// TwinCAT 3 PLC project Gearsim
// ProgramVersion: 3.1.4023.0
// libraries:
//   Struckig, * (Stefan Besler)
//   Tc3_Module, * (Beckhoff Automation GmbH)
//   ZApplication, 1.5.38.0 (Zeugwerk GmbH)
//   ZEquipment, 1.5.38.0 (Zeugwerk GmbH)
//   ZAux, 1.5.38.0 (Zeugwerk GmbH)
//   ZPlatform, 1.5.38.0 (Zeugwerk GmbH)
//   ZCore, 1.5.38.0 (Zeugwerk GmbH)
// project tree:
//   ZApp/App/ ZApp.TcPOU
//   ZApp/App/_DataTypes/ ZAppStep.TcDUT
//   ZApp/App/_States/ ZAppSequenceBoot.TcPOU, ZAppSequenceBootFault.TcPOU, ZAppSequenceRunning.TcPOU
//   ZApp/App/_SubObjects/ ZAppSequence.TcPOU
//   ZApp/Com/_DataTypes/ ZCom.TcDUT, ZComUnit.TcDUT
//   ZApp/Data/_DataTypes/ ZData.TcDUT, ZDataMachine.TcDUT, ZDataConfig.TcDUT, ZDataCalibration.TcDUT, ZDataRecipe.TcDUT
//   ZApp/Unit/Gear/ GearUnit.TcPOU, GearUnitProgram.TcPOU, IGear.TcIO
//   ZApp/Unit/Gear/_Com/ GearCom.TcDUT, GearComPublish.TcDUT, GearComPublishEquipment.TcDUT, GearComRef.TcDUT, GearComRequest.TcDUT, GearComSubscribe.TcDUT, GearComSubscribeEquipment.TcDUT
//   ZApp/Unit/Gear/_DataTypes/ GearRole.TcDUT, GearState.TcDUT, GearStep.TcDUT
//   ZApp/Unit/Gear/_Data/ GearDataCalibration.TcDUT, GearDataConfig.TcDUT, GearDataMachine.TcDUT, GearDataRef.TcDUT
//   ZApp/Unit/Gear/_Equipment/ GearActuator.TcPOU, GearAxis.TcPOU, GearEquipment.TcPOU, GearFieldbus.TcPOU, GearIo.TcPOU, GearLinkedUnit.TcPOU
//   ZApp/Unit/Gear/_States/ GearSequenceAutomatic.TcPOU, GearSequenceBoot.TcPOU, GearSequenceFaultReaction.TcPOU, GearSequenceGoHome.TcPOU, GearSequenceStop.TcPOU
//   ZApp/Unit/Gear/_SubObjects/ GearContainer.TcPOU, GearSequence.TcPOU
//   ZApp/Unit/Gear/_SubSequences/ GearSequenceAutomaticPrimary.TcPOU, GearSequenceAutomaticSecondarySimple.TcPOU, GearSequenceAutomaticSecondaryStruckig.TcPOU, GearSubSequence.TcPOU
//   ZApp/Unit/Machine/ IMachine.TcIO, MachineUnit.TcPOU, MachineUnitProgram.TcPOU
//   ZApp/Unit/Machine/_Com/ MachineCom.TcDUT, MachineComPublish.TcDUT, MachineComPublishEquipment.TcDUT, MachineComRef.TcDUT, MachineComRequest.TcDUT, MachineComSubscribe.TcDUT, MachineComSubscribeEquipment.TcDUT
//   ZApp/Unit/Machine/_DataTypes/ MachineState.TcDUT, MachineStep.TcDUT
//   ZApp/Unit/Machine/_Data/ MachineDataCalibration.TcDUT, MachineDataConfig.TcDUT, MachineDataMachine.TcDUT, MachineDataRef.TcDUT
//   ZApp/Unit/Machine/_Equipment/ MachineActuator.TcPOU, MachineAxis.TcPOU, MachineEquipment.TcPOU, MachineFieldbus.TcPOU, MachineIo.TcPOU, MachineLinkedUnit.TcPOU
//   ZApp/Unit/Machine/_States/ MachineSequenceAutomatic.TcPOU, MachineSequenceBoot.TcPOU, MachineSequenceFaultReaction.TcPOU, MachineSequenceGoHome.TcPOU, MachineSequenceStop.TcPOU
//   ZApp/Unit/Machine/_SubObjects/ MachineContainer.TcPOU, MachineSequence.TcPOU
//   ZApp/ ZGlobal.TcGVL, ZModuleProgram.TcPOU, ZModuleTask.TcTTO
// real-time tasks:
//   TASK ZModuleTask: cycle T#10ms, priority 20, ADS port 350
//   TASK ZModuleTask1: cycle T#10ms, priority 21, ADS port 351

CONFIGURATION Gearsim
    RESOURCE PLC ON TwinCAT3
        TASK ZModuleTask(INTERVAL := T#10ms, PRIORITY := 21);
        PROGRAM ZModuleProgram WITH ZModuleTask : ZModuleProgram;
    END_RESOURCE
END_CONFIGURATION

// ---- ZApp/App/_DataTypes/ZAppStep.TcDUT
{attribute 'qualified_only'}
{attribute 'to_string'}
TYPE ZAppStep :
(
  Undefined := 0
  
  ,BootBegin
  ,BootLoadDefaultData
  ,BootEnd
  ,BootFaultBegin
  ,BootFaultEnd 
  ,RunningBegin
  ,RunningEnd   
);
END_TYPE

// ---- ZApp/Com/_DataTypes/ZCom.TcDUT
TYPE ZCom :
STRUCT
  // module context
  App : ZApplication.ApplicationComPublish;
  Alarming : ZApplication.AlarmingCom;
  Messages : ZApplication.MessagingCom;
  
  // unit context
  Unit : ZComUnit;

END_STRUCT
END_TYPE

// ---- ZApp/Com/_DataTypes/ZComUnit.TcDUT
TYPE ZComUnit :
STRUCT
{region "LeftGear"}
{IF NOT (defined (LeftGear_disabled))}
  LeftGear : GearCom;
  {attribute 'ZId' := 'd1deea68-6f8b-4ea5-9916-7be69dc951fa'}
{END_IF}
{endregion}
{region "Machine"}
{IF NOT (defined (Machine_disabled))}
  Machine : MachineCom;
  {attribute 'ZId' := '9a1e8940-043c-4b8f-bd95-526fb267b71c'}
{END_IF}
{endregion}
{region "RightGear"}
{IF NOT (defined (RightGear_disabled))}
  RightGear : GearCom;
  {attribute 'ZId' := '215d1db4-d61a-4f46-91b5-612373b86c91'}
{END_IF}
{endregion}
{attribute '__ZwPlcApplicationComUnitDeclaration__'} // Do not remove this attribute! It is used for code generation.
END_STRUCT
END_TYPE

// ---- ZApp/Data/_DataTypes/ZData.TcDUT
TYPE ZData :
STRUCT
  Config : ZDataConfig;
  Machine : ZDataMachine;
  Calibration : ZDataCalibration;
  Recipe : ZDataRecipe;
END_STRUCT
END_TYPE

// ---- ZApp/Data/_DataTypes/ZDataMachine.TcDUT
TYPE ZDataMachine :
STRUCT
{region "PrimaryGear"}
{IF NOT (defined (PrimaryGear_disabled))}
  PrimaryGear : GearDataMachine;
  {attribute 'ZId' := 'd1deea68-6f8b-4ea5-9916-7be69dc951fa'}
{END_IF}
{endregion}
{region "Machine"}
{IF NOT (defined (Machine_disabled))}
  Machine : MachineDataMachine;
  {attribute 'ZId' := '9a1e8940-043c-4b8f-bd95-526fb267b71c'}
{END_IF}
{endregion}
{region "SimpleGear"}
{IF NOT (defined (SimpleGear_disabled))}
  SimpleGear : GearDataMachine;
  {attribute 'ZId' := '215d1db4-d61a-4f46-91b5-612373b86c91'}
{END_IF}
{endregion}
{region "StruckigGear"}
{IF NOT (defined (StruckigGear_disabled))}
  StruckigGear : GearDataMachine;
  {attribute 'ZId' := 'd827270e-999f-436d-80d5-b12442f5d1cf'}
{END_IF}
{endregion}
{attribute '__ZwPlcApplicationDataMachineDeclaration__'} // Do not remove this attribute! It is used for code generation.
END_STRUCT
END_TYPE

// ---- ZApp/Data/_DataTypes/ZDataConfig.TcDUT
TYPE ZDataConfig :
STRUCT
{region "PrimaryGear"}
{IF NOT (defined (PrimaryGear_disabled))}
  PrimaryGear : GearDataConfig;
  {attribute 'ZId' := 'd1deea68-6f8b-4ea5-9916-7be69dc951fa'}
{END_IF}
{endregion}
{region "Machine"}
{IF NOT (defined (Machine_disabled))}
  Machine : MachineDataConfig;
  {attribute 'ZId' := '9a1e8940-043c-4b8f-bd95-526fb267b71c'}
{END_IF}
{endregion}
{region "SimpleGear"}
{IF NOT (defined (SimpleGear_disabled))}
  SimpleGear : GearDataConfig;
  {attribute 'ZId' := '215d1db4-d61a-4f46-91b5-612373b86c91'}
{END_IF}
{endregion}
{region "StruckigGear"}
{IF NOT (defined (StruckigGear_disabled))}
  StruckigGear : GearDataConfig;
  {attribute 'ZId' := 'd827270e-999f-436d-80d5-b12442f5d1cf'}
{END_IF}
{endregion}
{attribute '__ZwPlcApplicationDataConfigDeclaration__'} // Do not remove this attribute! It is used for code generation.
END_STRUCT
END_TYPE

// ---- ZApp/Data/_DataTypes/ZDataCalibration.TcDUT
TYPE ZDataCalibration :
STRUCT
{region "PrimaryGear"}
{IF NOT (defined (PrimaryGear_disabled))}
  PrimaryGear : GearDataCalibration;
  {attribute 'ZId' := 'd1deea68-6f8b-4ea5-9916-7be69dc951fa'}
{END_IF}
{endregion}
{region "Machine"}
{IF NOT (defined (Machine_disabled))}
  Machine : MachineDataCalibration;
  {attribute 'ZId' := '9a1e8940-043c-4b8f-bd95-526fb267b71c'}
{END_IF}
{endregion}
{region "SimpleGear"}
{IF NOT (defined (SimpleGear_disabled))}
  SimpleGear : GearDataCalibration;
  {attribute 'ZId' := '215d1db4-d61a-4f46-91b5-612373b86c91'}
{END_IF}
{endregion}
{region "StruckigGear"}
{IF NOT (defined (StruckigGear_disabled))}
  StruckigGear : GearDataCalibration;
  {attribute 'ZId' := 'd827270e-999f-436d-80d5-b12442f5d1cf'}
{END_IF}
{endregion}
{attribute '__ZwPlcApplicationDataCalibrationDeclaration__'} // Do not remove this attribute! It is used for code generation.
END_STRUCT
END_TYPE

// ---- ZApp/Data/_DataTypes/ZDataRecipe.TcDUT
TYPE ZDataRecipe :
STRUCT
  RecipeParam1 : LREAL;
  RecipeParam2 : LREAL;
  RecipeParam3 : LREAL;
END_STRUCT
END_TYPE

// ---- ZApp/Unit/Gear/_Com/GearCom.TcDUT
/// This struct contains variables that
/// * are read from outside (e.g. HMI) to retrieve information about the unit's current state and (temporary) parameters (= `publish`) 
/// * are written from outside (e.g. HMI) to control the unit via ADS (= `subscribe`) 
TYPE GearCom :
STRUCT
  Publish : GearComPublish;
  Subscribe : GearComSubscribe;
END_STRUCT
END_TYPE

// ---- ZApp/Unit/Gear/_Com/GearComPublish.TcDUT
/// this is the container of informations that the unit wants to share with the world outside of the PLC
/// This struct should only be read from by external applications.
TYPE GearComPublish :
STRUCT
  State : ZApplication.UnitStateMachineState; // state the unit is in
  Request : GearComRequest; // booleans that indictate which action is currently possible to perform with this unit
  Equipment : GearComPublishEquipment;  // structs for equipment objects which are used by the bridges
END_STRUCT
END_TYPE

// ---- ZApp/Unit/Gear/_Com/GearComPublishEquipment.TcDUT
TYPE GearComPublishEquipment :
STRUCT

{region "PositionX : Axis"}
  PositionX : ZApplication.AxisComPublish;
  {attribute 'ZId' := 'fbe544fd-32f7-4a35-b34a-168d60744a34'}
{endregion}

{region "RotationC : Axis"}
  RotationC : ZApplication.AxisComPublish;
  {attribute 'ZId' := '01f1af52-e172-4e11-895e-2a66564d7b35'}
{endregion}

{attribute '__ZwPlcUnitComDeclaration__'} // Do not remove this attribute! It is used for code generation.

END_STRUCT
END_TYPE

// ---- ZApp/Unit/Gear/_Com/GearComRef.TcDUT
/// container for all communication data types that are used by the unit
TYPE GearComRef :
STRUCT
  Publish : REFERENCE TO GearComPublish; 
  Subscribe : REFERENCE TO GearComSubscribe; 
END_STRUCT
END_TYPE

// ---- ZApp/Unit/Gear/_Com/GearComRequest.TcDUT
TYPE GearComRequest :
STRUCT
  Start : BOOL;
  Stop : BOOL;
  GoHome : BOOL;
  Halt : BOOL;
END_STRUCT
END_TYPE

// ---- ZApp/Unit/Gear/_Com/GearComSubscribe.TcDUT
TYPE GearComSubscribe :
STRUCT
  Request : GearComRequest; // contains booleans that are used to start a specific sequence.
  Equipment : GearComSubscribeEquipment;  // structs for equipment objects which are used by the bridges
END_STRUCT
END_TYPE

// ---- ZApp/Unit/Gear/_Com/GearComSubscribeEquipment.TcDUT
TYPE GearComSubscribeEquipment :
STRUCT

{region "PositionX : Axis"}
  PositionX : ZApplication.AxisComSubscribe;
  {attribute 'ZId' := 'fbe544fd-32f7-4a35-b34a-168d60744a34'}
{endregion}

{region "RotationC : Axis"}
  RotationC : ZApplication.AxisComSubscribe;
  {attribute 'ZId' := '01f1af52-e172-4e11-895e-2a66564d7b35'}
{endregion}

{attribute '__ZwPlcUnitComDeclaration__'} // Do not remove this attribute! It is used for code generation.

END_STRUCT
END_TYPE

// ---- ZApp/Unit/Gear/_DataTypes/GearRole.TcDUT
{attribute 'qualified_only'}
{attribute 'strict'}
TYPE GearRole :
(
  Undefined
	,Primary
  ,SecondarySimple
  ,SecondaryStruckig
);
END_TYPE

// ---- ZApp/Unit/Gear/_DataTypes/GearState.TcDUT
/// This enumeration contains all used defined sequences of a unit.
/// Per default a unit makes use of the states that are contained in (UnitStateDefault)[xref:ZApplication.UnitStateDefault]. However,
/// most of the time a unit need to perform some application depend sequences that can be performed by putting the unit into userdefined states.
/// For instance, a robotic unit could use the state (automatic)[xref:ZApplication.UnitStateDefault] to lift an object from point A to point B,
/// a userdefined state could be used to open and close the robotic-units gripper, respectively
{attribute 'qualified_only'}
TYPE GearState :
(
	UserdefinedState1 := ZApplication.UnitStateMachineState.Last+1
);
END_TYPE

// ---- ZApp/Unit/Gear/_DataTypes/GearStep.TcDUT
/// This enumeration contains all steps that are used by the various sequences of a unit.
/// Sequences use a subrange (***Begin to ***End) of this enumeration.
{attribute 'qualified_only'}
{attribute 'to_string'}
TYPE GearStep :
(
  Undefined := 0
  
  ,BootBegin
  ,BootEnd 

  ,StopBegin
  ,StopEnd

  ,AutomaticBegin
  ,AutomaticEnd
  
  ,GoHomeBegin
  ,GoHomePositionX
  ,GoHomeRotationC
  ,GoHomeEnd 
  
  ,FaultReactionBegin
  ,FaultReactionEnd
  ,AutomaticPrimaryBegin
  ,AutomaticPrimaryHalt  
  ,AutomaticPrimaryEnd
  
  ,AutomaticSecondarySimpleBegin
  ,AutomaticSecondarySimpleCloseGap
  ,AutomaticSecondarySimpleSynchronized
  ,AutomaticSecondarySimpleOpenGap
  ,AutomaticSecondarySimpleTearDown
  ,AutomaticSecondarySimpleSpinFast
  ,AutomaticSecondarySimpleSpin
  ,AutomaticSecondarySimpleHalt    
  ,AutomaticSecondarySimpleEnd
  
  ,AutomaticSecondaryStruckigBegin
  ,AutomaticSecondaryStruckigRotate
  ,AutomaticSecondaryStruckigCloseGap
  ,AutomaticSecondaryStruckigSynchronized
  ,AutomaticSecondaryStruckigOpenGap
  ,AutomaticSecondaryStruckigTearDown
  ,AutomaticSecondaryStruckigSpinFast
  ,AutomaticSecondaryStruckigSpin
  ,AutomaticSecondaryStruckigHalt     
  ,AutomaticSecondaryStruckigEnd
);
END_TYPE

// ---- ZApp/Unit/Gear/_Data/GearDataCalibration.TcDUT
/// calibration that is determined by calibration sequences of the unit (static offsets, shifts)
TYPE GearDataCalibration :
STRUCT
  OffsetRotationC : LREAL;
END_STRUCT
END_TYPE

// ---- ZApp/Unit/Gear/_Data/GearDataConfig.TcDUT
/// configuration data that is used during boot to configure the Units equipment
TYPE GearDataConfig :
STRUCT
  Simulated : BOOL;
END_STRUCT
END_TYPE

// ---- ZApp/Unit/Gear/_Data/GearDataMachine.TcDUT
/// machine data that is used through most sequences of the unit (motor speed, axes positions, ...)
TYPE GearDataMachine :
STRUCT
  Role : GearRole;
  SlowspeedX : LREAL;
  HighspeedX : LREAL;
  HomePositionX : LREAL;
  SafePositionX : LREAL;
  SpinPositionX : LREAL;
  
  SlowspeedC : LREAL;
  HighspeedC : LREAL;  
  HomeRotationC : LREAL;
  
  ToothAngle : LREAL;
END_STRUCT
END_TYPE

// ---- ZApp/Unit/Gear/_Data/GearDataRef.TcDUT
/// container for all data that are used by the unit
TYPE GearDataRef :
STRUCT
  Config : REFERENCE TO GearDataConfig; // data required for booting the unit (axes configuration, simulation, parameters that have to be written in PREOP, ...)
  Machine : REFERENCE TO GearDataMachine; // speeds, positions, ...
  Calibration : REFERENCE TO GearDataCalibration; // offsets, shifts of nominal to actual values
END_STRUCT
END_TYPE

// ---- ZApp/Unit/Machine/_Com/MachineCom.TcDUT
/// This struct contains variables that
/// * are read from outside (e.g. HMI) to retrieve information about the unit's current state and (temporary) parameters (= `publish`) 
/// * are written from outside (e.g. HMI) to control the unit via ADS (= `subscribe`) 
TYPE MachineCom :
STRUCT
  Publish : MachineComPublish;
  Subscribe : MachineComSubscribe;
END_STRUCT
END_TYPE

// ---- ZApp/Unit/Machine/_Com/MachineComPublish.TcDUT
/// this is the container of informations that the unit wants to share with the world outside of the PLC
/// This struct should only be read from by external applications.
TYPE MachineComPublish :
STRUCT
  State : ZApplication.UnitStateMachineState; // state the unit is in
  Request : MachineComRequest; // booleans that indictate which action is currently possible to perform with this unit
  Equipment : MachineComPublishEquipment;  // structs for equipment objects which are used by the bridges
END_STRUCT
END_TYPE

// ---- ZApp/Unit/Machine/_Com/MachineComPublishEquipment.TcDUT
TYPE MachineComPublishEquipment :
STRUCT

{attribute '__ZwPlcUnitComDeclaration__'} // Do not remove this attribute! It is used for code generation.

END_STRUCT
END_TYPE

// ---- ZApp/Unit/Machine/_Com/MachineComRef.TcDUT
/// container for all communication data types that are used by the unit
TYPE MachineComRef :
STRUCT
  Publish : REFERENCE TO MachineComPublish; 
  Subscribe : REFERENCE TO MachineComSubscribe; 
END_STRUCT
END_TYPE

// ---- ZApp/Unit/Machine/_Com/MachineComRequest.TcDUT
TYPE MachineComRequest :
STRUCT
  Start : BOOL;
  Stop : BOOL;
  GoHome : BOOL;
  Halt : BOOL;
END_STRUCT
END_TYPE

// ---- ZApp/Unit/Machine/_Com/MachineComSubscribe.TcDUT
TYPE MachineComSubscribe :
STRUCT
  Request : MachineComRequest; // contains booleans that are used to start a specific sequence.
  Equipment : MachineComSubscribeEquipment;  // structs for equipment objects which are used by the bridges
END_STRUCT
END_TYPE

// ---- ZApp/Unit/Machine/_Com/MachineComSubscribeEquipment.TcDUT
TYPE MachineComSubscribeEquipment :
STRUCT

{attribute '__ZwPlcUnitComDeclaration__'} // Do not remove this attribute! It is used for code generation.

END_STRUCT
END_TYPE

// ---- ZApp/Unit/Machine/_DataTypes/MachineState.TcDUT
/// This enumeration contains all used defined sequences of a unit.
/// Per default a unit makes use of the states that are contained in (UnitStateDefault)[xref:ZApplication.UnitStateDefault]. However,
/// most of the time a unit need to perform some application depend sequences that can be performed by putting the unit into userdefined states.
/// For instance, a robotic unit could use the state (automatic)[xref:ZApplication.UnitStateDefault] to lift an object from point A to point B,
/// a userdefined state could be used to open and close the robotic-units gripper, respectively
{attribute 'qualified_only'}
TYPE MachineState :
(
	UserdefinedState1 := ZApplication.UnitStateMachineState.Last+1
);
END_TYPE

// ---- ZApp/Unit/Machine/_DataTypes/MachineStep.TcDUT
/// This enumeration contains all steps that are used by the various sequences of a unit.
/// Sequences use a subrange (***Begin to ***End) of this enumeration.
{attribute 'qualified_only'}
{attribute 'to_string'}
TYPE MachineStep :
(
  Undefined := 0
  
  ,BootBegin
  ,BootEnd 

  ,StopBegin
  ,StopEnd

  ,AutomaticBegin
  ,AutomaticEnd
  
  ,GoHomeBegin
  ,GoHomePositionX
  ,GoHomeRotationC
  ,GoHomeEnd 
  
  ,FaultReactionBegin
  ,FaultReactionEnd
);
END_TYPE

// ---- ZApp/Unit/Machine/_Data/MachineDataCalibration.TcDUT
/// calibration that is determined by calibration sequences of the unit (static offsets, shifts)
TYPE MachineDataCalibration :
STRUCT
END_STRUCT
END_TYPE

// ---- ZApp/Unit/Machine/_Data/MachineDataConfig.TcDUT
/// configuration data that is used during boot to configure the Units equipment
TYPE MachineDataConfig :
STRUCT
  Simulated : BOOL;
END_STRUCT
END_TYPE

// ---- ZApp/Unit/Machine/_Data/MachineDataMachine.TcDUT
/// machine data that is used through most sequences of the unit (motor speed, axes positions, ...)
TYPE MachineDataMachine :
STRUCT
  Slowspeed : LREAL;
  Highspeed : LREAL;
END_STRUCT
END_TYPE

// ---- ZApp/Unit/Machine/_Data/MachineDataRef.TcDUT
/// container for all data that are used by the unit
TYPE MachineDataRef :
STRUCT
  Config : REFERENCE TO MachineDataConfig; // data required for booting the unit (axes configuration, simulation, parameters that have to be written in PREOP, ...)
  Machine : REFERENCE TO MachineDataMachine; // speeds, positions, ...
  Calibration : REFERENCE TO MachineDataCalibration; // offsets, shifts of nominal to actual values
END_STRUCT
END_TYPE

// ---- ZApp/ZGlobal.TcGVL
{attribute 'qualified_only'}
VAR_GLOBAL
  Com : ZCom;
END_VAR
VAR_GLOBAL PERSISTENT
  Data : ZData;
END_VAR

// ---- ZApp/Unit/Gear/IGear.TcIO
INTERFACE IGear EXTENDS ZApplication.IUnit

PROPERTY InSpeed : BOOL
GET
END_GET
END_PROPERTY

PROPERTY PrimaryPositionC : LREAL
GET
END_GET
SET
END_SET
END_PROPERTY

PROPERTY PrimaryVelocityC : LREAL
GET
END_GET
SET
END_SET
END_PROPERTY

END_INTERFACE

// ---- ZApp/Unit/Machine/IMachine.TcIO
INTERFACE IMachine EXTENDS ZApplication.IUnit

END_INTERFACE

// ---- ZApp/ZModuleProgram.TcPOU
/// Zeugwerk Application
PROGRAM ZModuleProgram
VAR_INPUT
{region "ZModuleProgram : Utility"}
  App : ZApp(displayName:='Zeugwerk-Application Template', com:=ZGlobal.Com.App);
  Datetime : ZAux.DateTimeUM;
  {attribute 'ZId' := ''}
{endregion}
{region "ZModuleProgram : Logging"}
  Alarming : ZApplication.Alarming(App, datetime := Datetime, com := ZGlobal.Com.Alarming);
  LoggerHmi : ZApplication.Messaging(App, datetime := Datetime, com := ZGlobal.Com.Messages);
  LoggerFile : ZAux.LoggerFile7FF(App, datetime := Datetime, filePath:='C:\Zeugwerk\logs\messages.log', target:='');
  Logger : ZAux.Logging;
  {attribute 'ZId' := ''}
{endregion}  
{attribute '__ZwPlcApplicationModuleProgramDeclaration__'} // Do not remove this attribute! It is used for code generation.
{region "PrimaryGear"}
{undefine RunInSeparateProgram}
{IF NOT (defined (PrimaryGear_disabled)) AND NOT (defined (RunInSeparateProgram))}
  PrimaryGear : GearUnit(name := 'PrimaryGear', // name of the unit (for logging)
					  parent := App, // caller of the Unit's cyclic method. If the Unit runs in its own context use 0
						configdata := ZGlobal.Data.Config.PrimaryGear,
						machinedata := ZGlobal.Data.Machine.PrimaryGear,
						calibrationdata := ZGlobal.Data.Calibration.PrimaryGear,
						com := ZGlobal.Com.Unit.PrimaryGear);
  {attribute 'section' := '__ZwPlcUnitProgramDeclaration__'}
  {attribute 'ZId' := 'd1deea68-6f8b-4ea5-9916-7be69dc951fa'}
{END_IF}
{endregion}
{region "Machine"}
{undefine RunInSeparateProgram}
{IF NOT (defined (Machine_disabled)) AND NOT (defined (RunInSeparateProgram))}
  Machine : MachineUnit(name := 'Machine', // name of the unit (for logging)
					  parent := App, // caller of the Unit's cyclic method. If the Unit runs in its own context use 0
						configdata := ZGlobal.Data.Config.Machine,
						machinedata := ZGlobal.Data.Machine.Machine,
						calibrationdata := ZGlobal.Data.Calibration.Machine,
						com := ZGlobal.Com.Unit.Machine);
  {attribute 'section' := '__ZwPlcUnitProgramDeclaration__'}
  {attribute 'ZId' := '9a1e8940-043c-4b8f-bd95-526fb267b71c'}
{END_IF}
{endregion}
{region "SimpleGear"}
{undefine RunInSeparateProgram}
{IF NOT (defined (SimpleGear_disabled)) AND NOT (defined (RunInSeparateProgram))}
  SimpleGear : GearUnit(name := 'SimpleGear', // name of the unit (for logging)
					  parent := App, // caller of the Unit's cyclic method. If the Unit runs in its own context use 0
						configdata := ZGlobal.Data.Config.SimpleGear,
						machinedata := ZGlobal.Data.Machine.SimpleGear,
						calibrationdata := ZGlobal.Data.Calibration.SimpleGear,
						com := ZGlobal.Com.Unit.SimpleGear);
  {attribute 'section' := '__ZwPlcUnitProgramDeclaration__'}
  {attribute 'ZId' := '215d1db4-d61a-4f46-91b5-612373b86c91'}
{END_IF}
{endregion}
{region "StruckigGear"}
{undefine RunInSeparateProgram}
{IF NOT (defined (StruckigGear_disabled)) AND NOT (defined (RunInSeparateProgram))}
  StruckigGear : GearUnit(name := 'StruckigGear', // name of the unit (for logging)
					  parent := App, // caller of the Unit's cyclic method. If the Unit runs in its own context use 0
						configdata := ZGlobal.Data.Config.StruckigGear,
						machinedata := ZGlobal.Data.Machine.StruckigGear,
						calibrationdata := ZGlobal.Data.Calibration.StruckigGear,
						com := ZGlobal.Com.Unit.StruckigGear);
  {attribute 'section' := '__ZwPlcUnitProgramDeclaration__'}
  {attribute 'ZId' := 'd827270e-999f-436d-80d5-b12442f5d1cf'}
{END_IF}
{endregion}
{attribute '__ZwPlcUnitProgramDeclaration__'} // Do not remove this attribute! It is used for code generation.
END_VAR

{region "ZModuleProgram : Utility"}
  Datetime.Cyclic();
  App.Cyclic();
  {attribute 'ZId' := ''}
{endregion}
{attribute '__ZwPlcApplicationModuleProgramImplementation__'} // Do not remove this attribute! It is used for code generation.

END_PROGRAM

// ---- ZApp/App/ZApp.TcPOU
FUNCTION_BLOCK ZApp EXTENDS ZApplication.Application
VAR
  _boot : ZAppSequenceBoot;
  _bootFault : ZAppSequenceBootFault;
  _running : ZAppSequenceRunning;
END_VAR

METHOD FB_init : BOOL
VAR_INPUT
  bInitRetains : BOOL; /// if TRUE, the retain variables are initialized (warm start / cold start)
  bInCopyCode : BOOL; /// if TRUE, the instance afterwards gets moved into the copy code (online change)
  displayName : ZCore.ZString;
  com : REFERENCE TO ZApplication.ApplicationComPublish;
END_VAR
SetBootSequence(_boot);
SetBootFaultSequence(_bootFault);
SetRunningSequence(_running);
END_METHOD

END_FUNCTION_BLOCK

// ---- ZApp/App/_States/ZAppSequenceBoot.TcPOU
FUNCTION_BLOCK ZAppSequenceBoot EXTENDS ZAppSequence IMPLEMENTS ZCore.ISequence
VAR
  _step : ZCore.Step(ZAppStep.BootBegin, ZAppStep.BootEnd);
END_VAR

IF OnStart(_step)
THEN
  // init custom sequence variables here ...
END_IF

REPEAT
  LogStep();

  CASE _step.Index OF
    (* -------------------------------------------------------------------------------------------------------------------------------- *)
    ZAppStep.BootBegin:
    (* -------------------------------------------------------------------------------------------------------------------------------- *)
    
      IF _step.OnEntry()
      THEN
        ZModuleProgram.LoggerFile.MinimumLevel := ZCore.LogLevel.Trace;
        ZModuleProgram.Logger.AddLogger(ZModuleProgram.LoggerFile);        
        {attribute '__ZwPlcAppZComModuleContext__'} // Do not remove this attribute! It is used for code generation.      
      END_IF
      
	  IF ZModuleProgram.Datetime.State <> ZCore.ObjectState.Booting
      THEN
        _step.SetNext(ZAppStep.BootLoadDefaultData);        
      END_IF
      
    (* -------------------------------------------------------------------------------------------------------------------------------- *)
    ZAppStep.BootLoadDefaultData:
    (* -------------------------------------------------------------------------------------------------------------------------------- *)

      LoadDefaultConfigData();
      
      IF IsCommissioning()
      THEN
        LoadDefaultData();
      END_IF
      
      _step.SetNext(ZAppStep.BootEnd);
      
    (* -------------------------------------------------------------------------------------------------------------------------------- *)
    ZAppStep.BootEnd:
    (* -------------------------------------------------------------------------------------------------------------------------------- *)
      SetBusy(FALSE);
      
  ELSE
    Abort('sequence contains unhandled step');
  END_CASE
UNTIL _step.IsNotRepeatable() OR_ELSE NOT Busy END_REPEAT

METHOD  IsCommissioning : BOOL
IsCommissioning := TRUE;
END_METHOD

METHOD FINAL LoadDefaultConfigData

{region "PrimaryGear"}
  {IF NOT (defined (PrimaryGear_disabled))}
  ZGlobal.Data.Config.PrimaryGear.Simulated := TRUE;
  {region "UserInitCode"}
  // put your individual init code for this unit here
  {endregion}
  {END_IF}
  {attribute 'ZId' := 'd1deea68-6f8b-4ea5-9916-7be69dc951fa'}
{endregion}

{region "Machine"}
  {IF NOT (defined (Machine_disabled))}
  ZGlobal.Data.Config.Machine.Simulated := TRUE;
  {region "UserInitCode"}
  // put your individual init code for this unit here
  {endregion}
  {END_IF}
  {attribute 'ZId' := '9a1e8940-043c-4b8f-bd95-526fb267b71c'}
{endregion}

{region "SimpleGear"}
  {IF NOT (defined (SimpleGear_disabled))}
  ZGlobal.Data.Config.SimpleGear.Simulated := TRUE;
  {region "UserInitCode"}
  // put your individual init code for this unit here
  {endregion}
  {END_IF}
  {attribute 'ZId' := '215d1db4-d61a-4f46-91b5-612373b86c91'}
{endregion}

{region "StruckigGear"}
  {IF NOT (defined (StruckigGear_disabled))}
  ZGlobal.Data.Config.StruckigGear.Simulated := TRUE;
  {region "UserInitCode"}
  // put your individual init code for this unit here
  {endregion}
  {END_IF}
  {attribute 'ZId' := 'd827270e-999f-436d-80d5-b12442f5d1cf'}
{endregion}

{attribute '__ZwPlcUnitLoadDefaultConfigData__'} // Do not remove this attribute! It is used for code generation.
END_METHOD

METHOD FINAL LoadDefaultData
ZGlobal.Data.Machine.PrimaryGear.Role := GearRole.Primary;
ZGlobal.Data.Machine.PrimaryGear.SlowspeedX := 200;
ZGlobal.Data.Machine.PrimaryGear.HighspeedX := 500;
ZGlobal.Data.Machine.PrimaryGear.HomePositionX := 0;
ZGlobal.Data.Machine.PrimaryGear.SafePositionX := 0;
ZGlobal.Data.Machine.PrimaryGear.SpinPositionX := 0;
ZGlobal.Data.Machine.PrimaryGear.SlowspeedC := 15;
ZGlobal.Data.Machine.PrimaryGear.HighspeedC := 30;
ZGlobal.Data.Machine.PrimaryGear.ToothAngle := 360.0 / 32.0;
ZGlobal.Data.Calibration.PrimaryGear.OffsetRotationC := 0;

ZGlobal.Data.Machine.SimpleGear.Role := GearRole.SecondarySimple;
ZGlobal.Data.Machine.SimpleGear.SlowspeedX := 200;
ZGlobal.Data.Machine.SimpleGear.HighspeedX := 500;
ZGlobal.Data.Machine.SimpleGear.HomePositionX := -30;
ZGlobal.Data.Machine.SimpleGear.SafePositionX := -30;
ZGlobal.Data.Machine.SimpleGear.SpinPositionX := -160;
ZGlobal.Data.Machine.SimpleGear.SlowspeedC := 15;
ZGlobal.Data.Machine.SimpleGear.HighspeedC := 30;
ZGlobal.Data.Machine.SimpleGear.ToothAngle := ZGlobal.Data.Machine.PrimaryGear.ToothAngle;
ZGlobal.Data.Calibration.SimpleGear.OffsetRotationC := ZGlobal.Data.Machine.StruckigGear.ToothAngle / 2;

ZGlobal.Data.Machine.StruckigGear.Role := GearRole.SecondaryStruckig;
ZGlobal.Data.Machine.StruckigGear.SlowspeedX := 200;
ZGlobal.Data.Machine.StruckigGear.HighspeedX := 500;
ZGlobal.Data.Machine.StruckigGear.HomePositionX := -10;
ZGlobal.Data.Machine.StruckigGear.SafePositionX := -10;
ZGlobal.Data.Machine.StruckigGear.SpinPositionX := -160;
ZGlobal.Data.Machine.StruckigGear.SlowspeedC := 15;
ZGlobal.Data.Machine.StruckigGear.HighspeedC := 30;
ZGlobal.Data.Machine.StruckigGear.ToothAngle := ZGlobal.Data.Machine.PrimaryGear.ToothAngle;
ZGlobal.Data.Calibration.StruckigGear.OffsetRotationC := ZGlobal.Data.Machine.StruckigGear.ToothAngle / 2;

{attribute '__ZwPlcUnitLoadDefaultData__'} // Do not remove this attribute! It is used for code generation.
END_METHOD

END_FUNCTION_BLOCK

// ---- ZApp/App/_SubObjects/ZAppSequence.TcPOU
FUNCTION_BLOCK ABSTRACT ZAppSequence EXTENDS ZApplication.Sequence IMPLEMENTS ZCore.ISequence

METHOD StepDecoded : ZCore.ZString
VAR_INPUT
  stepIndex : INT;
END_VAR
VAR_INST
  _stepIndexDecoded : ZAppStep;
END_VAR
_stepIndexDecoded := stepIndex;
StepDecoded := TO_STRING(_stepIndexDecoded);
END_METHOD

END_FUNCTION_BLOCK

// ---- ZApp/App/_States/ZAppSequenceBootFault.TcPOU
FUNCTION_BLOCK ZAppSequenceBootFault EXTENDS ZAppSequence IMPLEMENTS ZCore.ISequence
VAR
  _step : ZCore.Step(ZAppStep.BootFaultBegin, ZAppStep.BootFaultEnd);
END_VAR

IF OnStart(_step)
THEN
  // init custom sequence variables here ...
END_IF

REPEAT
  LogStep();

  CASE _step.Index OF
    (* -------------------------------------------------------------------------------------------------------------------------------- *)
    ZAppStep.BootFaultBegin:
    (* -------------------------------------------------------------------------------------------------------------------------------- *)
      _step.SetNext(ZAppStep.BootFaultEnd);
      
    (* -------------------------------------------------------------------------------------------------------------------------------- *)
    ZAppStep.BootFaultEnd:
    (* -------------------------------------------------------------------------------------------------------------------------------- *)
      SetBusy(FALSE);
      
  ELSE
    Abort('sequence contains unhandled step');
  END_CASE
UNTIL _step.IsNotRepeatable() OR_ELSE NOT Busy END_REPEAT

END_FUNCTION_BLOCK

// ---- ZApp/App/_States/ZAppSequenceRunning.TcPOU
FUNCTION_BLOCK ZAppSequenceRunning EXTENDS ZAppSequence IMPLEMENTS ZCore.ISequence
VAR
  _step : ZCore.Step(ZAppStep.RunningBegin, ZAppStep.RunningEnd);
END_VAR

IF OnStart(_step)
THEN
  // init custom sequence variables here ...
END_IF

REPEAT
  LogStep();

  CASE _step.Index OF
    (* -------------------------------------------------------------------------------------------------------------------------------- *)
    ZAppStep.RunningBegin:
    (* -------------------------------------------------------------------------------------------------------------------------------- *)
      ; // implement me
      
    (* -------------------------------------------------------------------------------------------------------------------------------- *)
    ZAppStep.RunningEnd:
    (* -------------------------------------------------------------------------------------------------------------------------------- *)
      SetBusy(FALSE);
      
  ELSE
    Abort('sequence contains unhandled step');
  END_CASE
UNTIL _step.IsNotRepeatable() OR_ELSE NOT Busy END_REPEAT

END_FUNCTION_BLOCK

// ---- ZApp/Unit/Gear/GearUnit.TcPOU
/// Declaration of a distinct unit of this application
FUNCTION_BLOCK GearUnit EXTENDS ZApplication.Unit IMPLEMENTS IGear
VAR
  _equipment : GearEquipment(THIS^);
  _data : GearDataRef;
  _com : GearComRef;

  _boot : GearSequenceBoot(THIS^);
  _automatic : GearSequenceAutomatic(THIS^);
  _stop : GearSequenceStop(THIS^);
  _gohome : GearSequenceGoHome(THIS^);
  _faultReaction : GearSequenceFaultReaction(THIS^);
  
  _statemachine : ZApplication.UnitStateMachine;
  _subSequence : GearSubSequence(THIS^);

  _observeTimer : ZAux.Timer;
END_VAR

{attribute 'ZId' := '4c08bcb1-14c0-4e8f-9942-ed50c5db2fbe'}

IF _observeTimer.Done THEN
  _observeTimer.WaitAsync(0.1);
  
  // monitor _com for requested actions (e.g. start homing, start automatic mode, ...)
  ObserveRequest(_com.Subscribe.Request.Start, ZApplication.UnitStateMachineState.Automatic);
  ObserveRequest(_com.Subscribe.Request.Stop, ZApplication.UnitStateMachineState.Stop);
  ObserveRequest(_com.Subscribe.Request.GoHome, ZApplication.UnitStateMachineState.GoHome);
  ObserveRequest(_com.Subscribe.Request.Halt, ZApplication.UnitStateMachineState.Halt);
  
  // provide relevant information via ADS
  _com.Publish.Request.Stop := _stateMachine.IsTransitionAllowed(ZApplication.UnitStateMachineState.Stop);
  _com.Publish.Request.Start := _stateMachine.IsTransitionAllowed(ZApplication.UnitStateMachineState.Automatic);
  _com.Publish.Request.GoHome := _stateMachine.IsTransitionAllowed(ZApplication.UnitStateMachineState.GoHome);
  _com.Publish.Request.Halt := _stateMachine.IsTransitionAllowed(ZApplication.UnitStateMachineState.Halt);

  _com.Publish.State := _stateMachine.State();
END_IF

METHOD FB_init : BOOL
VAR_INPUT
  bInitRetains : BOOL; // if TRUE, the retain variables are initialized (warm start / cold start)
  bInCopyCode : BOOL;  // if TRUE, the instance afterwards gets moved into the copy code (online change)
  parent : ZCore.IManagedObject; // caller of the Unit's cyclic method. If the Unit runs in its own context use 0
  name : ZCore.ZString;  // name of this unit as it should show up in the logger
  configdata : REFERENCE TO GearDataConfig;  // reference to the configuration data that is used during boot to configure the Units equipment
  machinedata : REFERENCE TO GearDataMachine; // reference to the machine data that is used through most sequences of the unit (motor speed, axes positions, ...)
  calibrationdata : REFERENCE TO GearDataCalibration;  // reference to calibration that is determined by calibration sequences of the unit (static offsets, shifts)
  com : REFERENCE TO GearCom;  // reference to the communication interface that is used to control this Unit via ADS
END_VAR
_name := name;

// initialize local logger decorator
_loggerDecorator.FB_init(bInitRetains, bInCopyCode, name, ZModuleProgram.Logger);
_alarmingDecorator.FB_init(bInitRetains, bInCopyCode, name, ZModuleProgram.Alarming);

// setup data
_data.Config REF= configdata;
_data.Machine REF= machinedata;
_data.Calibration REF= calibrationdata;
_com.Publish REF= com.Publish;
_com.Subscribe REF= com.Subscribe;

// ------- sequence initialization, map sequences of this unit to the statemachine -------
{attribute '__ZwPlcUnitInitSequenceImplementation__'} // Do not remove this attribute! It is used for code generation.
_statemachine.SetSequence(ZApplication.UnitStateMachineState.Boot, _boot);
_statemachine.SetSequence(ZApplication.UnitStateMachineState.FaultReaction, _faultReaction);
_statemachine.SetSequence(ZApplication.UnitStateMachineState.Gohome, _gohome);
_statemachine.SetSequence(ZApplication.UnitStateMachineState.Stop, _stop);
_statemachine.SetSequence(ZApplication.UnitStateMachineState.Automatic, _automatic);

_statemachine.SetName(_name);
_statemachine.SetLogger(_logger);

// set initial state
_statemachine.SetState(ZApplication.UnitStateMachineState.Boot);
SetStateMachine(_statemachine);
END_METHOD

END_FUNCTION_BLOCK

// ---- ZApp/Unit/Gear/_Equipment/GearEquipment.TcPOU
/// This function block is a container for equipment that is used by this unit.
/// Equipment is grouped by its kind (actuator, axes, io, ...).
/// It extends from [ManagedObjectContainer](xref:ZCore.ManagedObjectContainer) such that the parent
/// (= the unit itself) can be passed to equipment instances.
FUNCTION_BLOCK GearEquipment EXTENDS GearContainer
VAR_INPUT
  Io : GearIo(_parent);
  Actuator : GearActuator(_parent);
  Axis : GearAxis(_parent);
  Fieldbus : GearFieldbus(_parent);
  Unit : GearLinkedUnit(_parent);
END_VAR

END_FUNCTION_BLOCK

// ---- ZApp/Unit/Gear/_SubObjects/GearContainer.TcPOU
FUNCTION_BLOCK GearContainer EXTENDS ZCore.ObjectContainer
VAR_INPUT
END_VAR
VAR_OUTPUT
END_VAR
VAR
  {attribute 'hide'}
  _parent : REFERENCE TO GearUnit;
END_VAR

{attribute 'hide' }
METHOD FB_init : BOOL
VAR_INPUT
	bInitRetains : BOOL; // if TRUE, the retain variables are initialized (warm start / cold start)
	bInCopyCode : BOOL;  // if TRUE, the instance afterwards gets moved into the copy code (online change)
  unit : REFERENCE TO GearUnit;
END_VAR
_parent REF= unit;
END_METHOD

END_FUNCTION_BLOCK

// ---- ZApp/Unit/Gear/_Equipment/GearIo.TcPOU
/// This function block is a container for all I/Os that are used by this unit.
/// The parent of all objects can be directly transfered in their constructor (this is only relevant for equipment objects
/// that have to be managed (e.g. [DebouncedInput](xref:ZEquipment.DebouncedInput), [Light](xref:ZEquipment.Light), ...).
FUNCTION_BLOCK GearIo EXTENDS GearContainer
VAR
  {attribute 'hide'}
  _iobridge : ZApplication.IoBridge(_parent);
END_VAR
VAR_INPUT

{attribute '__ZwPlcUnitEquipmentDeclaration__'} // Do not remove this attribute! It is used for code generation.
END_VAR

IF _isInitialized
THEN
  RETURN;
END_IF

  _iobridge.SetLogger(_parent._logger);

{attribute '__ZwPlcUnitEquipmentImplementation__'} // Do not remove this attribute! It is used for code generation.

_isInitialized := TRUE;

END_FUNCTION_BLOCK

// ---- ZApp/Unit/Gear/_Equipment/GearActuator.TcPOU
/// This function block is a container for all actuator objects that are used by this unit.
/// The parent of all objects can be directly transfered in their constructor (this is only relevant for equipment objects
/// that have to be managed (e.g. [DebouncedInput](xref:ZEquipment.DebouncedInput), [Light](xref:ZEquipment.Light), ...).
FUNCTION_BLOCK GearActuator EXTENDS GearContainer
VAR
  {attribute 'hide'}
  _actuatorbridge : ZApplication.ActuatorBridge(_parent);
  {attribute 'hide'}
  _iobridge : ZApplication.IoBridge(_parent);
END_VAR
VAR_INPUT

{attribute '__ZwPlcUnitEquipmentDeclaration__'} // Do not remove this attribute! It is used for code generation.
END_VAR

IF _isInitialized
THEN
  RETURN;
END_IF

  _actuatorbridge.SetLogger(_parent._logger);

{attribute '__ZwPlcUnitEquipmentImplementation__'} // Do not remove this attribute! It is used for code generation.

_isInitialized := TRUE;

END_FUNCTION_BLOCK

// ---- ZApp/Unit/Gear/_Equipment/GearAxis.TcPOU
/// This function block is a container for all axis objects that are used by this unit.
/// The parent of all objects can be directly transfered in their constructor (this is only relevant for equipment objects
/// that have to be managed (e.g. [DebouncedInput](xref:ZEquipment.DebouncedInput), [Light](xref:ZEquipment.Light), ...).
FUNCTION_BLOCK GearAxis EXTENDS GearContainer
VAR
  {attribute 'hide'}
  _axisbridge : ZApplication.AxisBridge(_parent);
END_VAR
VAR_INPUT

{region "PositionX : AxisPlcOpenMc"}
  PositionX : ZEquipment.AxisSimulated(_parent);
  {attribute 'ZId' := 'fbe544fd-32f7-4a35-b34a-168d60744a34'}
{endregion}

{region "RotationC : AxisPlcOpenMc"}
  RotationC : ZEquipment.AxisSimulated(_parent);
  {attribute 'ZId' := '01f1af52-e172-4e11-895e-2a66564d7b35'}
{endregion}

{attribute '__ZwPlcUnitEquipmentDeclaration__'} // Do not remove this attribute! It is used for code generation.
END_VAR

IF _isInitialized
THEN
  RETURN;
END_IF

  _axisbridge.SetLogger(_parent._logger);

{region "PositionX : AxisPlcOpenMc"}
  PositionX.SetLogger(_parent._logger);
  PositionX.SetName(name:='PositionX');
  PositionX.SetSimulation(_parent._data.Config.Simulated);
  _axisbridge.WithHoming(PositionX)
     .WithMovePosition(PositionX)
     .WithMoveVelocity(PositionX)
     .WithHalt(PositionX)
     .WithVelocityFeedrate(PositionX)
     .WithFeedbackPosition(PositionX)
     .WithFeedbackVelocity(PositionX)
     .WithFeedbackCurrent(PositionX)
     .AddAxis (axis:=PositionX, publish:=_parent._com.Publish.Equipment.PositionX, subscribe:=_parent._com.Subscribe.Equipment.PositionX);

  {region "UserInitCode"}
  // put your individual init code for this Axis here
  {endregion}

  {attribute 'ZId' := 'fbe544fd-32f7-4a35-b34a-168d60744a34'}
{endregion}

{region "RotationC : AxisPlcOpenMc"}
  RotationC.SetLogger(_parent._logger);
  RotationC.SetName(name:='RotationC');
  RotationC.SetSimulation(_parent._data.Config.Simulated);
  _axisbridge.WithHoming(RotationC)
     .WithMovePosition(RotationC)
     .WithMoveVelocity(RotationC)
     .WithHalt(RotationC)
     .WithVelocityFeedrate(RotationC)
     .WithFeedbackPosition(RotationC)
     .WithFeedbackVelocity(RotationC)
     .WithFeedbackCurrent(RotationC)
     .AddAxis (axis:=RotationC, publish:=_parent._com.Publish.Equipment.RotationC, subscribe:=_parent._com.Subscribe.Equipment.RotationC);	   
			
  {region "UserInitCode"}
  // put your individual init code for this Axis here
  {endregion}

  {attribute 'ZId' := '01f1af52-e172-4e11-895e-2a66564d7b35'}
{endregion}

{attribute '__ZwPlcUnitEquipmentImplementation__'} // Do not remove this attribute! It is used for code generation.

_isInitialized := TRUE;

END_FUNCTION_BLOCK

// ---- ZApp/Unit/Gear/_Equipment/GearFieldbus.TcPOU
/// This function block is a container for all axis objects that are used by this unit.
/// The parent of all objects can be directly transfered in their constructor (this is only relevant for equipment objects
/// that have to be managed (e.g. [DebouncedInput](xref:ZEquipment.DebouncedInput), [Light](xref:ZEquipment.Light), ...).
FUNCTION_BLOCK GearFieldbus EXTENDS GearContainer
VAR
END_VAR
VAR_INPUT

{attribute '__ZwPlcUnitEquipmentDeclaration__'} // Do not remove this attribute! It is used for code generation.
END_VAR

IF _isInitialized
THEN
  RETURN;
END_IF

{attribute '__ZwPlcUnitEquipmentImplementation__'} // Do not remove this attribute! It is used for code generation.

_isInitialized := TRUE;

END_FUNCTION_BLOCK

// ---- ZApp/Unit/Gear/_Equipment/GearLinkedUnit.TcPOU
/// This function block is a container for all linked units that are used by this unit.
/// Linked units can be addressed through their individual interface.
FUNCTION_BLOCK GearLinkedUnit EXTENDS GearContainer
VAR_INPUT

{attribute '__ZwPlcUnitEquipmentDeclaration__'} // Do not remove this attribute! It is used for code generation.
END_VAR

IF _isInitialized
THEN
  RETURN;
END_IF

{attribute '__ZwPlcUnitEquipmentImplementation__'} // Do not remove this attribute! It is used for code generation.

_isInitialized := TRUE;

END_FUNCTION_BLOCK

// ---- ZApp/Unit/Gear/_States/GearSequenceBoot.TcPOU
FUNCTION_BLOCK GearSequenceBoot EXTENDS GearSequence IMPLEMENTS ZCore.ISequence
VAR
  _step : ZCore.Step(GearStep.BootBegin, GearStep.BootEnd);
END_VAR

IF OnStart(_step) THEN
  ; // init custom sequence variables here ...
END_IF

REPEAT
  LogStep();

  CASE _step.Index OF
    (* -------------------------------------------------------------------------------------------------------------------------------- *)
    GearStep.BootBegin:
    (* -------------------------------------------------------------------------------------------------------------------------------- *)
      IF _step.OnEntry()
      THEN
        // initialize subsequences
        _subSequence();

        // initialize equipment
        _io();
        _actuator();
        _fieldbus();
        _axis();
        _unit();
      END_IF
      
      _parent._objectManager.Cyclic();      
      Assert(_parent._objectManager);
      IF _parent._objectManager.Booted
      THEN
        _step.SetNext(GearStep.BootEnd);
      END_IF

    (* -------------------------------------------------------------------------------------------------------------------------------- *)
    GearStep.BootEnd:
    (* -------------------------------------------------------------------------------------------------------------------------------- *)
      SetBusy(FALSE);
      
  ELSE
    Abort('sequence contains unhandled step');
  END_CASE
UNTIL _step.IsNotRepeatable() OR_ELSE NOT Busy END_REPEAT

END_FUNCTION_BLOCK

// ---- ZApp/Unit/Gear/_SubObjects/GearSequence.TcPOU
FUNCTION_BLOCK GearSequence EXTENDS ZApplication.Sequence
VAR
  {attribute 'hide'}
  _parent : REFERENCE TO GearUnit;
  _io : REFERENCE TO GearIo;
  _actuator : REFERENCE TO GearActuator;
  _fieldbus : REFERENCE TO GearFieldbus;
  _axis : REFERENCE TO GearAxis;
  _data : REFERENCE TO GearDataRef;
  _unit : REFERENCE TO GearLinkedUnit;  
END_VAR

METHOD FB_init : BOOL
VAR_INPUT
  bInitRetains : BOOL; // if TRUE, the retain variables are initialized (warm start / cold start)
  bInCopyCode : BOOL;  // if TRUE, the instance afterwards gets moved into the copy code (online change)
  unit : REFERENCE TO GearUnit;
END_VAR
_parent REF= unit;
_alarming := unit._alarming;
_io REF= unit._equipment.Io;
_actuator REF= unit._equipment.Actuator;
_fieldbus REF= unit._equipment.Fieldbus;
_axis REF= unit._equipment.Axis;
_unit REF= unit._equipment.Unit;
_data REF= unit._data;
_loggerDiagnostics.SetLogger(unit._logger);
END_METHOD

METHOD StepDecoded : ZCore.ZString
VAR_INPUT
  stepIndex : INT;
END_VAR
VAR_INST
  _stepIndexDecoded : GearStep;
END_VAR
_stepIndexDecoded := stepIndex;
stepDecoded := TO_STRING(_stepIndexDecoded);
END_METHOD

END_FUNCTION_BLOCK

// ---- ZApp/Unit/Gear/_States/GearSequenceAutomatic.TcPOU
FUNCTION_BLOCK GearSequenceAutomatic EXTENDS GearSequence IMPLEMENTS ZCore.ISequence
VAR
  _step : ZCore.Step(GearStep.AutomaticBegin, GearStep.AutomaticEnd);
  _sequence : ZCore.ISequence;
END_VAR

IF NOT Busy THEN
  RETURN;
END_IF

IF OnStart(_step) THEN
  ; // init custom sequence variables here ...
END_IF

IF OnStop() THEN
  RETURN; // external stop was triggered
END_IF

IF OnHalt() THEN
  Halting := TRUE;
END_IF

REPEAT
  LogStep();

  CASE _step.Index OF
    (* -------------------------------------------------------------------------------------------------------------------------------- *)
    GearStep.AutomaticBegin:
    (* -------------------------------------------------------------------------------------------------------------------------------- *)
      IF _step.OnEntry()
      THEN
        CASE _data.Machine.Role
        OF
          GearRole.Primary: _sequence := _subSequence.AutomaticPrimary;
          GearRole.SecondarySimple: _sequence := _subSequence.AutomaticSecondarySimple;
          GearRole.SecondaryStruckig: _sequence := _subSequence.AutomaticSecondaryStruckig;
        ELSE
          Abort('Role not implemented!');
          RETURN;
				END_CASE
        
        _sequence.RunAsync(THIS^);
      END_IF

      _sequence.Cyclic();
      Await(obj1:=_sequence, nextStep:=GearStep.AutomaticEnd);
      
    (* -------------------------------------------------------------------------------------------------------------------------------- *)
    GearStep.AutomaticEnd:
    (* -------------------------------------------------------------------------------------------------------------------------------- *)
      SetBusy(FALSE);
  
  ELSE
    Abort('sequence contains unhandled step');
  END_CASE
UNTIL _step.IsNotRepeatable() OR_ELSE NOT Busy END_REPEAT

END_FUNCTION_BLOCK

// ---- ZApp/Unit/Gear/_States/GearSequenceStop.TcPOU
FUNCTION_BLOCK GearSequenceStop EXTENDS GearSequence IMPLEMENTS ZCore.ISequence
VAR
  _step : ZCore.Step(GearStep.StopBegin, GearStep.StopEnd);
  _timerSim : ZAux.Timer;
END_VAR

IF OnStart(_step) THEN
  ; // init custom sequence variables here ...
END_IF

REPEAT
  LogStep();

  CASE _step.Index OF
    (* -------------------------------------------------------------------------------------------------------------------------------- *)
    GearStep.StopBegin:
    (* -------------------------------------------------------------------------------------------------------------------------------- *)
      IF _step.OnEntry()
      THEN
        _axis.PositionX.StopAsync(THIS^);
        _axis.RotationC.StopAsync(THIS^);
      END_IF
      
      Await2( _axis.PositionX, _axis.RotationC, nextStep:=GearStep.StopEnd);

    (* -------------------------------------------------------------------------------------------------------------------------------- *)
    GearStep.StopEnd:
    (* -------------------------------------------------------------------------------------------------------------------------------- *)    
      SetBusy(FALSE);
  
  ELSE
    Abort('sequence contains unhandled step');
  END_CASE
UNTIL _step.IsNotRepeatable() OR_ELSE NOT Busy END_REPEAT

END_FUNCTION_BLOCK

// ---- ZApp/Unit/Gear/_States/GearSequenceGoHome.TcPOU
FUNCTION_BLOCK GearSequenceGoHome EXTENDS GearSequence IMPLEMENTS ZCore.ISequence
VAR
  _step : ZCore.Step(GearStep.GohomeBegin, GearStep.GohomeEnd);
  _timer : ZAux.Timer;
END_VAR

IF NOT Busy THEN
  RETURN;
END_IF

IF OnStart(_step) THEN
  ; // init custom sequence variables here ...
END_IF

IF OnStop() THEN
  RETURN; // external stop was triggered
END_IF

IF OnHalt() THEN
  ; // Halting := TRUE; // Uncomment to acknowledge that the sequence is halting
END_IF

REPEAT
  LogStep();

  CASE _step.Index OF
    (* -------------------------------------------------------------------------------------------------------------------------------- *)
    GearStep.GoHomeBegin:
    (* -------------------------------------------------------------------------------------------------------------------------------- *)

      _step.SetNext(index:=GearStep.GoHomePositionX);

	(* -------------------------------------------------------------------------------------------------------------------------------- *)
    GearStep.GoHomePositionX:
    (* -------------------------------------------------------------------------------------------------------------------------------- *)
      IF _step.OnEntry()
      THEN        
        _axis.PositionX.MoveAbsoluteAsync(THIS^, _data.Machine.HomePositionX, _data.Machine.SlowspeedX);
      END_IF
      
      Await(obj1:=_axis.PositionX, nextStep:=GearStep.GoHomeRotationC);

	(* -------------------------------------------------------------------------------------------------------------------------------- *)
    GearStep.GoHomeRotationC:
    (* -------------------------------------------------------------------------------------------------------------------------------- *)
      IF _step.OnEntry()
      THEN        
        _axis.RotationC.MoveAbsoluteAsync(THIS^,
            _axis.RotationC.ActualPosition - _parent.PhaseOffsetC + _data.Machine.ToothAngle, _data.Machine.SlowspeedC);
      END_IF
      
      Await(obj1:=_axis.PositionX, nextStep:=GearStep.GoHomeEnd);

    (* -------------------------------------------------------------------------------------------------------------------------------- *)
    GearStep.GoHomeEnd:
    (* -------------------------------------------------------------------------------------------------------------------------------- *)
      SetBusy(FALSE);
  
  ELSE
    Abort('sequence contains unhandled step');
  END_CASE
UNTIL _step.IsNotRepeatable() OR_ELSE NOT Busy END_REPEAT

END_FUNCTION_BLOCK

// ---- ZApp/Unit/Gear/_States/GearSequenceFaultReaction.TcPOU
FUNCTION_BLOCK GearSequenceFaultReaction EXTENDS GearSequence IMPLEMENTS ZCore.ISequence
VAR
  _step : ZCore.Step(GearStep.FaultReactionBegin, GearStep.FaultReactionEnd);
  _timerSim : ZAux.Timer;
END_VAR

IF OnStart(_step) THEN
  ; // init custom sequence variables here ...
END_IF

REPEAT
  LogStep();

  CASE _step.Index OF
    (* -------------------------------------------------------------------------------------------------------------------------------- *)
    GearStep.FaultReactionBegin:
    (* -------------------------------------------------------------------------------------------------------------------------------- *)
      IF _step.OnEntry()
      THEN
        _axis.PositionX.StopAsync(THIS^);
        _axis.RotationC.StopAsync(THIS^);
      END_IF
      
      _step.SetNext(GearStep.FaultReactionEnd);

    (* -------------------------------------------------------------------------------------------------------------------------------- *)
    GearStep.FaultReactionEnd:
    (* -------------------------------------------------------------------------------------------------------------------------------- *)    
      SetBusy(FALSE);
  
  ELSE
    Abort('sequence contains unhandled step');
  END_CASE
UNTIL _step.IsNotRepeatable() OR_ELSE NOT Busy END_REPEAT

END_FUNCTION_BLOCK

// ---- ZApp/Unit/Gear/_SubSequences/GearSubSequence.TcPOU
FUNCTION_BLOCK GearSubSequence EXTENDS GearContainer
VAR_INPUT

{region "fc3b2a3d-8136-4db1-aaab-6cca602a7edf"}
  AutomaticPrimary : GearSequenceAutomaticPrimary(_parent);
{endregion} // #fc3b2a3d-8136-4db1-aaab-6cca602a7edf
{region "16b36b8d-fde6-4830-a9e3-c3507d13faec"}
  AutomaticSecondarySimple : GearSequenceAutomaticSecondarySimple(_parent);
{endregion} // #16b36b8d-fde6-4830-a9e3-c3507d13faec
{region "79362472-a44e-4c7c-b677-cada7c3c933b"}
  AutomaticSecondaryStruckig : GearSequenceAutomaticSecondaryStruckig(_parent);
{endregion} // #79362472-a44e-4c7c-b677-cada7c3c933b
  {attribute '__ZwPlcUnitSequence__'}
  
END_VAR

IF NOT _isInitialized THEN
  
{region "fc3b2a3d-8136-4db1-aaab-6cca602a7edf"}
  AutomaticPrimary.SetName('AutomaticPrimary');
  AutomaticPrimary.SetLogger(_parent._logger);
{endregion} // #fc3b2a3d-8136-4db1-aaab-6cca602a7edf
{region "16b36b8d-fde6-4830-a9e3-c3507d13faec"}
  AutomaticSecondarySimple.SetName('AutomaticSecondarySimple');
  AutomaticSecondarySimple.SetLogger(_parent._logger);
{endregion} // #16b36b8d-fde6-4830-a9e3-c3507d13faec
{region "79362472-a44e-4c7c-b677-cada7c3c933b"}
  AutomaticSecondaryStruckig.SetName('AutomaticSecondaryStruckig');
  AutomaticSecondaryStruckig.SetLogger(_parent._logger);
{endregion} // #79362472-a44e-4c7c-b677-cada7c3c933b
  {attribute '__ZwPlcUnitSequence__'}
  
  _isInitialized := TRUE;

END_IF

END_FUNCTION_BLOCK

// ---- ZApp/Unit/Gear/_SubSequences/GearSequenceAutomaticPrimary.TcPOU
FUNCTION_BLOCK GearSequenceAutomaticPrimary EXTENDS GearSequence IMPLEMENTS ZCore.ISequence
VAR
  _step : ZCore.Step(GearStep.AutomaticPrimaryBegin, GearStep.AutomaticPrimaryEnd);
END_VAR

IF NOT Busy THEN
  RETURN;
END_IF

IF OnStart(_step) THEN
  ; // init custom sequence variables here ...
END_IF

IF OnStop() THEN
  RETURN; // external stop was triggered
END_IF

IF OnHalt() THEN
  Halting := TRUE;
END_IF

REPEAT
  LogStep();

  CASE _step.Index OF
    (* -------------------------------------------------------------------------------------------------------------------------------- *)
    GearStep.AutomaticPrimaryBegin:
    (* -------------------------------------------------------------------------------------------------------------------------------- *)
      IF _step.OnEntry()
      THEN
        _axis.RotationC.MoveVelocityAsync(THIS^, _data.Machine.HighspeedC);
      END_IF

      IF Halting
      THEN
        _step.SetNext(GearStep.AutomaticPrimaryHalt);
			END_IF
      
    (* -------------------------------------------------------------------------------------------------------------------------------- *)
    GearStep.AutomaticPrimaryHalt:
    (* -------------------------------------------------------------------------------------------------------------------------------- *)    
      IF _step.OnEntry()
      THEN
        _axis.RotationC.StopAsync(THIS^);
      END_IF

      Assert(_axis.RotationC);
      Await(obj1:=_axis.RotationC, nextStep:=GearStep.AutomaticPrimaryEnd);
            
    (* -------------------------------------------------------------------------------------------------------------------------------- *)
    GearStep.AutomaticPrimaryEnd:
    (* -------------------------------------------------------------------------------------------------------------------------------- *)
      SetBusy(FALSE);
  
  ELSE
    Abort('sequence contains unhandled step');
  END_CASE
UNTIL _step.IsNotRepeatable() OR_ELSE NOT Busy END_REPEAT

END_FUNCTION_BLOCK

// ---- ZApp/Unit/Gear/_SubSequences/GearSequenceAutomaticSecondarySimple.TcPOU
FUNCTION_BLOCK GearSequenceAutomaticSecondarySimple EXTENDS GearSequence IMPLEMENTS ZCore.ISequence
VAR
  _step : ZCore.Step(GearStep.AutomaticSecondarySimpleBegin, GearStep.AutomaticSecondarySimpleEnd);
  _timer : ZAux.Timer;
  _waitDurationShort : ZAux.RandomGaussian(seed:=0, mu:=0.5, sigma:=1);
  _waitDurationLong : ZAux.RandomGaussian(seed:=0, mu:=3, sigma:=1);
  _spin : ZAux.RandomUniform(seed:=0, low:=0, high:=1);  
END_VAR

IF NOT Busy THEN
  RETURN;
END_IF

IF OnStart(_step) THEN
  ; // init custom sequence variables here ...
END_IF

IF OnStop() THEN
  RETURN; // external stop was triggered
END_IF

IF OnHalt() THEN
  ; // Halting := TRUE; // Uncomment to acknowledge that the sequence is halting
END_IF

REPEAT
  LogStep();

  CASE _step.Index OF
    (* -------------------------------------------------------------------------------------------------------------------------------- *)
    GearStep.AutomaticSecondarySimpleBegin:
    (* -------------------------------------------------------------------------------------------------------------------------------- *)
      IF _step.OnEntry()
      THEN
        _waitDurationShort.SetSeed(_data.Machine.Role);
        _waitDurationLong.SetSeed(_data.Machine.Role);

        _axis.PositionX.MoveAbsoluteAsync(THIS^, _data.Machine.SafePositionX, _data.Machine.HighspeedX);
        _axis.RotationC.MoveVelocityAsync(THIS^, _data.Machine.HighspeedC);
      END_IF

      Await2(obj1:=_axis.RotationC, obj2:=_axis.PositionX, nextStep:=GearStep.AutomaticSecondarySimpleCloseGap);
      
    (* -------------------------------------------------------------------------------------------------------------------------------- *)
    GearStep.AutomaticSecondarySimpleCloseGap:
    (* -------------------------------------------------------------------------------------------------------------------------------- *)
      IF _step.OnEntry()
      THEN
        _axis.PositionX.MoveAbsoluteAsync(THIS^, _data.Machine.SpinPositionX, _data.Machine.HighspeedX);
      END_IF

      Assert(_axis.RotationC);
      Await(obj1:=_axis.PositionX, nextStep:=GearStep.AutomaticSecondarySimpleSynchronized);
      _step.SetNext(GearStep.AutomaticSecondarySimpleSynchronized);   
      
    (* -------------------------------------------------------------------------------------------------------------------------------- *)
    GearStep.AutomaticSecondarySimpleSynchronized:
    (* -------------------------------------------------------------------------------------------------------------------------------- *)
    
      IF _step.OnEntry()
      THEN
        _timer.WaitAsync(_waitDurationLong.Next());
      END_IF
    
      Assert(_axis.PositionX);
      Assert(_axis.RotationC);
      
      IF _timer.Done
      THEN
        IF _spin.Next() > 0.5
        THEN
          _step.SetNext(GearStep.AutomaticSecondarySimpleOpenGap);
				END_IF
			END_IF
      
      IF Halting
      THEN
        _step.SetNext(GearStep.AutomaticSecondarySimpleOpenGap);  
			END_IF
    
    (* -------------------------------------------------------------------------------------------------------------------------------- *)
    GearStep.AutomaticSecondarySimpleOpenGap:
    (* -------------------------------------------------------------------------------------------------------------------------------- *)    
      IF _step.OnEntry()
      THEN
        _axis.PositionX.MoveAbsoluteAsync(THIS^, _data.Machine.SafePositionX, _data.Machine.HighspeedX);
      END_IF

      Assert(_axis.RotationC);
      
      IF Halting
      THEN
        Await(obj1:=_axis.PositionX, nextStep:=GearStep.AutomaticSecondarySimpleTearDown);
        _step.SetNext(GearStep.AutomaticSecondarySimpleEnd);
      ELSE
        _step.SetNext(GearStep.AutomaticSecondarySimpleSpinFast);
			END_IF

    (* -------------------------------------------------------------------------------------------------------------------------------- *)
    GearStep.AutomaticSecondarySimpleSpinFast:
    (* -------------------------------------------------------------------------------------------------------------------------------- *)
      IF _step.OnEntry()
      THEN
        _timer.WaitAsync(_waitDurationLong.Next());
        _axis.RotationC.MoveVelocityAsync(THIS^, _data.Machine.HighspeedC*2);
      END_IF

      Assert(_axis.RotationC);

      IF _timer.Done
      THEN
        _step.SetNext(GearStep.AutomaticSecondarySimpleSpin);          
			END_IF


    (* -------------------------------------------------------------------------------------------------------------------------------- *)
    GearStep.AutomaticSecondarySimpleSpin:
    (* -------------------------------------------------------------------------------------------------------------------------------- *)
      IF _step.OnEntry()
      THEN
        _timer.WaitAsync(_waitDurationShort.Next());
        _axis.RotationC.MoveVelocityAsync(THIS^, _data.Machine.HighspeedC);
      END_IF

      Assert(_axis.RotationC);
      
      IF _timer.Done
      THEN
        _step.SetNext(GearStep.AutomaticSecondarySimpleCloseGap);          
			END_IF
      
    (* -------------------------------------------------------------------------------------------------------------------------------- *)
    GearStep.AutomaticSecondarySimpleTearDown:
    (* -------------------------------------------------------------------------------------------------------------------------------- *)    
      IF _step.OnEntry()
      THEN
        _axis.PositionX.MoveAbsoluteAsync(THIS^, _data.Machine.HomePositionX, _data.Machine.HighspeedX);
        _axis.RotationC.MoveVelocityAsync(THIS^, _data.Machine.SlowspeedC);
      END_IF

      Assert(_axis.RotationC);
      _step.SetNext(GearStep.AutomaticSecondarySimpleHalt);
      
    (* -------------------------------------------------------------------------------------------------------------------------------- *)
    GearStep.AutomaticSecondarySimpleHalt:
    (* -------------------------------------------------------------------------------------------------------------------------------- *)    
      IF _step.OnEntry()
      THEN
        _axis.RotationC.StopAsync(THIS^);
      END_IF

      Assert(_axis.RotationC);
      Await(obj1:=_axis.RotationC, nextStep:=GearStep.AutomaticSecondarySimpleEnd);
      
    (* -------------------------------------------------------------------------------------------------------------------------------- *)
    GearStep.AutomaticSecondarySimpleEnd:
    (* -------------------------------------------------------------------------------------------------------------------------------- *)
      SetBusy(FALSE);
  
  ELSE
    Abort('sequence contains unhandled step');
  END_CASE
UNTIL _step.IsNotRepeatable() OR_ELSE NOT Busy END_REPEAT

END_FUNCTION_BLOCK

// ---- ZApp/Unit/Gear/_SubSequences/GearSequenceAutomaticSecondaryStruckig.TcPOU
FUNCTION_BLOCK GearSequenceAutomaticSecondaryStruckig EXTENDS GearSequence IMPLEMENTS ZCore.ISequence
VAR
  _step : ZCore.Step(GearStep.AutomaticSecondaryStruckigBegin, GearStep.AutomaticSecondaryStruckigEnd);
  _timer : ZAux.Timer;
  _waitDurationShort : ZAux.RandomGaussian(seed:=0, mu:=0.5, sigma:=1);
  _waitDurationLong : ZAux.RandomGaussian(seed:=0, mu:=3, sigma:=1);
  _spin : ZAux.RandomUniform(seed:=0, low:=0, high:=1);  
END_VAR

IF NOT Busy THEN
  RETURN;
END_IF

IF OnStart(_step) THEN
  ; // init custom sequence variables here ...
END_IF

IF OnStop() THEN
  RETURN; // external stop was triggered
END_IF

IF OnHalt() THEN
  ; // Halting := TRUE; // Uncomment to acknowledge that the sequence is halting
END_IF

REPEAT
  LogStep();

  CASE _step.Index OF
    (* -------------------------------------------------------------------------------------------------------------------------------- *)
    GearStep.AutomaticSecondaryStruckigBegin:
    (* -------------------------------------------------------------------------------------------------------------------------------- *)
      IF _step.OnEntry()
      THEN
        _waitDurationShort.SetSeed(_data.Machine.Role);
        _waitDurationLong.SetSeed(_data.Machine.Role);
      
        _axis.PositionX.MoveAbsoluteAsync(THIS^, _data.Machine.SafePositionX, _data.Machine.HighspeedX);
        _axis.RotationC.MoveVelocityAsync(THIS^, _data.Machine.HighspeedC);
      END_IF

      _step.SetNext(GearStep.AutomaticSecondaryStruckigCloseGap);
      
    (* -------------------------------------------------------------------------------------------------------------------------------- *)
    GearStep.AutomaticSecondaryStruckigCloseGap:
    (* -------------------------------------------------------------------------------------------------------------------------------- *)
      IF _step.OnEntry()
      THEN
        _axis.PositionX.MoveAbsoluteAsync(THIS^, _data.Machine.SpinPositionX, _data.Machine.HighspeedX);
      END_IF

      Assert(_axis.RotationC);
      Await(obj1:=_axis.PositionX, nextStep:=GearStep.AutomaticSecondaryStruckigSynchronized);
      _step.SetNext(GearStep.AutomaticSecondaryStruckigSynchronized);   
      
    (* -------------------------------------------------------------------------------------------------------------------------------- *)
    GearStep.AutomaticSecondaryStruckigSynchronized:
    (* -------------------------------------------------------------------------------------------------------------------------------- *)
    
      IF _step.OnEntry()
      THEN
        _timer.WaitAsync(_waitDurationLong.Next());
			END_IF
    
      Assert(_axis.PositionX);
      Assert(_axis.RotationC);
      
      IF _timer.Done
      THEN
        IF _spin.Next() > 0.5
        THEN
          _step.SetNext(GearStep.AutomaticSecondaryStruckigOpenGap);
				END_IF
			END_IF
      
      IF Halting
      THEN
        _step.SetNext(GearStep.AutomaticSecondaryStruckigOpenGap);  
			END_IF
    
    (* -------------------------------------------------------------------------------------------------------------------------------- *)
    GearStep.AutomaticSecondaryStruckigOpenGap:
    (* -------------------------------------------------------------------------------------------------------------------------------- *)    
      IF _step.OnEntry()
      THEN
        _axis.PositionX.MoveAbsoluteAsync(THIS^, _data.Machine.SafePositionX, _data.Machine.HighspeedX);
      END_IF

      Assert(_axis.RotationC);
      
      IF Halting
      THEN
        Await(obj1:=_axis.PositionX, nextStep:=GearStep.AutomaticSecondaryStruckigTearDown);
        _step.SetNext(GearStep.AutomaticSecondaryStruckigEnd);
      ELSE
        _step.SetNext(GearStep.AutomaticSecondaryStruckigSpinFast);
			END_IF

    (* -------------------------------------------------------------------------------------------------------------------------------- *)
    GearStep.AutomaticSecondaryStruckigSpinFast:
    (* -------------------------------------------------------------------------------------------------------------------------------- *)
      IF _step.OnEntry()
      THEN
        _timer.WaitAsync(_waitDurationLong.Next());
        _axis.RotationC.MoveVelocityAsync(THIS^, _data.Machine.HighspeedC*2);
      END_IF

      Assert(_axis.RotationC);

      IF _timer.Done
      THEN
        _step.SetNext(GearStep.AutomaticSecondaryStruckigSpin);          
			END_IF


    (* -------------------------------------------------------------------------------------------------------------------------------- *)
    GearStep.AutomaticSecondaryStruckigSpin:
    (* -------------------------------------------------------------------------------------------------------------------------------- *)
      IF _step.OnEntry()
      THEN
        _timer.WaitAsync(_waitDurationShort.Next());
        _axis.RotationC.MoveVelocityAsync(THIS^, _data.Machine.HighspeedC);
      END_IF

      Assert(_axis.RotationC);
      
      IF _timer.Done
      THEN
        _step.SetNext(GearStep.AutomaticSecondaryStruckigCloseGap);          
			END_IF
      
    (* -------------------------------------------------------------------------------------------------------------------------------- *)
    GearStep.AutomaticSecondaryStruckigTearDown:
    (* -------------------------------------------------------------------------------------------------------------------------------- *)    
      IF _step.OnEntry()
      THEN
        _axis.PositionX.MoveAbsoluteAsync(THIS^, _data.Machine.HomePositionX, _data.Machine.HighspeedX);
        _axis.RotationC.MoveVelocityAsync(THIS^, _data.Machine.SlowspeedC);
      END_IF

      Assert(_axis.RotationC);
      _step.SetNext(GearStep.AutomaticSecondaryStruckigEnd);
      
    (* -------------------------------------------------------------------------------------------------------------------------------- *)
    GearStep.AutomaticSecondaryStruckigHalt:
    (* -------------------------------------------------------------------------------------------------------------------------------- *)    
      IF _step.OnEntry()
      THEN
        _axis.RotationC.StopAsync(THIS^);
      END_IF

      Assert(_axis.RotationC);
      Await(obj1:=_axis.RotationC, nextStep:=GearStep.AutomaticSecondaryStruckigEnd);
      
    (* -------------------------------------------------------------------------------------------------------------------------------- *)
    GearStep.AutomaticSecondaryStruckigEnd:
    (* -------------------------------------------------------------------------------------------------------------------------------- *)
      SetBusy(FALSE);
  
  ELSE
    Abort('sequence contains unhandled step');
  END_CASE
UNTIL _step.IsNotRepeatable() OR_ELSE NOT Busy END_REPEAT

END_FUNCTION_BLOCK

// ---- ZApp/Unit/Machine/MachineUnit.TcPOU
/// Declaration of a distinct unit of this application
FUNCTION_BLOCK MachineUnit EXTENDS ZApplication.Unit IMPLEMENTS IMachine
VAR
  _equipment : MachineEquipment(THIS^);
  _data : MachineDataRef;
  _com : MachineComRef;

  _boot : MachineSequenceBoot(THIS^);
  _automatic : MachineSequenceAutomatic(THIS^);
  _stop : MachineSequenceStop(THIS^);
  _gohome : MachineSequenceGoHome(THIS^);
  _faultReaction : MachineSequenceFaultReaction(THIS^);
  
  _statemachine : ZApplication.UnitStateMachine;

  _observeTimer : ZAux.Timer;
END_VAR

{attribute 'ZId' := '5918240d-d585-4361-8bfb-e76d2a3c3fb9'}

_equipment.Unit.SimpleGear.PrimaryPositionC := _equipment.Unit.PrimaryGear.PrimaryPositionC;
_equipment.Unit.SimpleGear.PrimaryVelocityC := _equipment.Unit.PrimaryGear.PrimaryVelocityC;
_equipment.Unit.StruckigGear.PrimaryPositionC := _equipment.Unit.PrimaryGear.PrimaryPositionC;
_equipment.Unit.StruckigGear.PrimaryVelocityC := _equipment.Unit.PrimaryGear.PrimaryVelocityC;

IF _observeTimer.Done THEN
  _observeTimer.WaitAsync(0.1);
  
  // monitor _com for requested actions (e.g. start homing, start automatic mode, ...)
  ObserveRequest(_com.Subscribe.Request.Start, ZApplication.UnitStateMachineState.Automatic);
  ObserveRequest(_com.Subscribe.Request.Stop, ZApplication.UnitStateMachineState.Stop);
  ObserveRequest(_com.Subscribe.Request.GoHome, ZApplication.UnitStateMachineState.GoHome);
  ObserveRequest(_com.Subscribe.Request.Halt, ZApplication.UnitStateMachineState.Halt);
  
  // provide relevant information via ADS
  _com.Publish.Request.Stop := _stateMachine.IsTransitionAllowed(ZApplication.UnitStateMachineState.Stop);
  _com.Publish.Request.Start := _stateMachine.IsTransitionAllowed(ZApplication.UnitStateMachineState.Automatic);
  _com.Publish.Request.GoHome := _stateMachine.IsTransitionAllowed(ZApplication.UnitStateMachineState.GoHome);
  _com.Publish.Request.Halt := _stateMachine.IsTransitionAllowed(ZApplication.UnitStateMachineState.Halt);

  _com.Publish.State := _stateMachine.State();
END_IF

METHOD FB_init : BOOL
VAR_INPUT
  bInitRetains : BOOL; // if TRUE, the retain variables are initialized (warm start / cold start)
  bInCopyCode : BOOL;  // if TRUE, the instance afterwards gets moved into the copy code (online change)
  parent : ZCore.IManagedObject; // caller of the Unit's cyclic method. If the Unit runs in its own context use 0
  name : ZCore.ZString;  // name of this unit as it should show up in the logger
  configdata : REFERENCE TO MachineDataConfig;  // reference to the configuration data that is used during boot to configure the Units equipment
  machinedata : REFERENCE TO MachineDataMachine; // reference to the machine data that is used through most sequences of the unit (motor speed, axes positions, ...)
  calibrationdata : REFERENCE TO MachineDataCalibration;  // reference to calibration that is determined by calibration sequences of the unit (static offsets, shifts)
  com : REFERENCE TO MachineCom;  // reference to the communication interface that is used to control this Unit via ADS
END_VAR
_name := name;

// initialize local logger decorator
_loggerDecorator.FB_init(bInitRetains, bInCopyCode, name, ZModuleProgram.Logger);
_alarmingDecorator.FB_init(bInitRetains, bInCopyCode, name, ZModuleProgram.Alarming);

// setup data
_data.Config REF= configdata;
_data.Machine REF= machinedata;
_data.Calibration REF= calibrationdata;
_com.Publish REF= com.Publish;
_com.Subscribe REF= com.Subscribe;

// ------- sequence initialization, map sequences of this unit to the statemachine -------
{attribute '__ZwPlcUnitInitSequenceImplementation__'} // Do not remove this attribute! It is used for code generation.
_statemachine.SetSequence(ZApplication.UnitStateMachineState.Boot, _boot);
_statemachine.SetSequence(ZApplication.UnitStateMachineState.FaultReaction, _faultReaction);
_statemachine.SetSequence(ZApplication.UnitStateMachineState.Gohome, _gohome);
_statemachine.SetSequence(ZApplication.UnitStateMachineState.Stop, _stop);
_statemachine.SetSequence(ZApplication.UnitStateMachineState.Automatic, _automatic);

_statemachine.SetName(_name);
_statemachine.SetLogger(_logger);

// set initial state
_statemachine.SetState(ZApplication.UnitStateMachineState.Boot);
SetStateMachine(_statemachine);
END_METHOD

END_FUNCTION_BLOCK

// ---- ZApp/Unit/Machine/_Equipment/MachineEquipment.TcPOU
/// This function block is a container for equipment that is used by this unit.
/// Equipment is grouped by its kind (actuator, axes, io, ...).
/// It extends from [ManagedObjectContainer](xref:ZCore.ManagedObjectContainer) such that the parent
/// (= the unit itself) can be passed to equipment instances.
FUNCTION_BLOCK MachineEquipment EXTENDS MachineContainer
VAR_INPUT
  Io : MachineIo(_parent);
  Actuator : MachineActuator(_parent);
  Axis : MachineAxis(_parent);
  Fieldbus : MachineFieldbus(_parent);
  Unit : MachineLinkedUnit(_parent);
END_VAR

END_FUNCTION_BLOCK

// ---- ZApp/Unit/Machine/_SubObjects/MachineContainer.TcPOU
FUNCTION_BLOCK MachineContainer EXTENDS ZCore.ObjectContainer
VAR_INPUT
END_VAR
VAR_OUTPUT
END_VAR
VAR
  {attribute 'hide'}
  _parent : REFERENCE TO MachineUnit;
END_VAR

{attribute 'hide' }
METHOD FB_init : BOOL
VAR_INPUT
	bInitRetains : BOOL; // if TRUE, the retain variables are initialized (warm start / cold start)
	bInCopyCode : BOOL;  // if TRUE, the instance afterwards gets moved into the copy code (online change)
  unit : REFERENCE TO MachineUnit;
END_VAR
_parent REF= unit;
END_METHOD

END_FUNCTION_BLOCK

// ---- ZApp/Unit/Machine/_Equipment/MachineIo.TcPOU
/// This function block is a container for all I/Os that are used by this unit.
/// The parent of all objects can be directly transfered in their constructor (this is only relevant for equipment objects
/// that have to be managed (e.g. [DebouncedInput](xref:ZEquipment.DebouncedInput), [Light](xref:ZEquipment.Light), ...).
FUNCTION_BLOCK MachineIo EXTENDS MachineContainer
VAR
  {attribute 'hide'}
  _iobridge : ZApplication.IoBridge(_parent);
END_VAR
VAR_INPUT

{attribute '__ZwPlcUnitEquipmentDeclaration__'} // Do not remove this attribute! It is used for code generation.
END_VAR

IF _isInitialized
THEN
  RETURN;
END_IF

  _iobridge.SetLogger(_parent._logger);

{attribute '__ZwPlcUnitEquipmentImplementation__'} // Do not remove this attribute! It is used for code generation.

_isInitialized := TRUE;

END_FUNCTION_BLOCK

// ---- ZApp/Unit/Machine/_Equipment/MachineActuator.TcPOU
/// This function block is a container for all actuator objects that are used by this unit.
/// The parent of all objects can be directly transfered in their constructor (this is only relevant for equipment objects
/// that have to be managed (e.g. [DebouncedInput](xref:ZEquipment.DebouncedInput), [Light](xref:ZEquipment.Light), ...).
FUNCTION_BLOCK MachineActuator EXTENDS MachineContainer
VAR
  {attribute 'hide'}
  _actuatorbridge : ZApplication.ActuatorBridge(_parent);
  {attribute 'hide'}
  _iobridge : ZApplication.IoBridge(_parent);
END_VAR
VAR_INPUT

{attribute '__ZwPlcUnitEquipmentDeclaration__'} // Do not remove this attribute! It is used for code generation.
END_VAR

IF _isInitialized
THEN
  RETURN;
END_IF

  _actuatorbridge.SetLogger(_parent._logger);

{attribute '__ZwPlcUnitEquipmentImplementation__'} // Do not remove this attribute! It is used for code generation.

_isInitialized := TRUE;

END_FUNCTION_BLOCK

// ---- ZApp/Unit/Machine/_Equipment/MachineAxis.TcPOU
/// This function block is a container for all axis objects that are used by this unit.
/// The parent of all objects can be directly transfered in their constructor (this is only relevant for equipment objects
/// that have to be managed (e.g. [DebouncedInput](xref:ZEquipment.DebouncedInput), [Light](xref:ZEquipment.Light), ...).
FUNCTION_BLOCK MachineAxis EXTENDS MachineContainer
VAR
  {attribute 'hide'}
  _axisbridge : ZApplication.AxisBridge(_parent);
END_VAR
VAR_INPUT

{attribute '__ZwPlcUnitEquipmentDeclaration__'} // Do not remove this attribute! It is used for code generation.
END_VAR

IF _isInitialized
THEN
  RETURN;
END_IF

  _axisbridge.SetLogger(_parent._logger);

{attribute '__ZwPlcUnitEquipmentImplementation__'} // Do not remove this attribute! It is used for code generation.

_isInitialized := TRUE;

END_FUNCTION_BLOCK

// ---- ZApp/Unit/Machine/_Equipment/MachineFieldbus.TcPOU
/// This function block is a container for all axis objects that are used by this unit.
/// The parent of all objects can be directly transfered in their constructor (this is only relevant for equipment objects
/// that have to be managed (e.g. [DebouncedInput](xref:ZEquipment.DebouncedInput), [Light](xref:ZEquipment.Light), ...).
FUNCTION_BLOCK MachineFieldbus EXTENDS MachineContainer
VAR
END_VAR
VAR_INPUT

{attribute '__ZwPlcUnitEquipmentDeclaration__'} // Do not remove this attribute! It is used for code generation.
END_VAR

IF _isInitialized
THEN
  RETURN;
END_IF

{attribute '__ZwPlcUnitEquipmentImplementation__'} // Do not remove this attribute! It is used for code generation.

_isInitialized := TRUE;

END_FUNCTION_BLOCK

// ---- ZApp/Unit/Machine/_Equipment/MachineLinkedUnit.TcPOU
/// This function block is a container for all linked units that are used by this unit.
/// Linked units can be addressed through their individual interface.
FUNCTION_BLOCK MachineLinkedUnit EXTENDS MachineContainer
VAR_INPUT
  PrimaryGear : IGear;
  SimpleGear : IGear; 
  StruckigGear : IGear;  
 
{attribute '__ZwPlcUnitEquipmentDeclaration__'} // Do not remove this attribute! It is used for code generation.
END_VAR

IF _isInitialized
THEN
  RETURN;
END_IF

PrimaryGear := ZModuleProgram.PrimaryGear;
SimpleGear := ZModuleProgram.SimpleGear;
StruckigGear := ZModuleProgram.StruckigGear;


{attribute '__ZwPlcUnitEquipmentImplementation__'} // Do not remove this attribute! It is used for code generation.

_isInitialized := TRUE;

END_FUNCTION_BLOCK

// ---- ZApp/Unit/Machine/_States/MachineSequenceBoot.TcPOU
FUNCTION_BLOCK MachineSequenceBoot EXTENDS MachineSequence IMPLEMENTS ZCore.ISequence
VAR
  _step : ZCore.Step(MachineStep.BootBegin, MachineStep.BootEnd);
END_VAR

IF OnStart(_step) THEN
  ; // init custom sequence variables here ...
END_IF

REPEAT
  LogStep();

  CASE _step.Index OF
    (* -------------------------------------------------------------------------------------------------------------------------------- *)
    MachineStep.BootBegin:
    (* -------------------------------------------------------------------------------------------------------------------------------- *)
      IF _step.OnEntry()
      THEN
        // initialize equipment
        _io();
        _actuator();
        _fieldbus();
        _axis();
        _unit();
      END_IF
      
      _parent._objectManager.Cyclic();      
      Assert(_parent._objectManager);
      IF _parent._objectManager.Booted
      THEN
        _step.SetNext(MachineStep.BootEnd);
      END_IF

    (* -------------------------------------------------------------------------------------------------------------------------------- *)
    MachineStep.BootEnd:
    (* -------------------------------------------------------------------------------------------------------------------------------- *)
      SetBusy(FALSE);
      
  ELSE
    Abort('sequence contains unhandled step');
  END_CASE
UNTIL _step.IsNotRepeatable() OR_ELSE NOT Busy END_REPEAT

END_FUNCTION_BLOCK

// ---- ZApp/Unit/Machine/_SubObjects/MachineSequence.TcPOU
FUNCTION_BLOCK MachineSequence EXTENDS ZApplication.Sequence
VAR
  {attribute 'hide'}
  _parent : REFERENCE TO MachineUnit;
  _io : REFERENCE TO MachineIo;
  _actuator : REFERENCE TO MachineActuator;
  _fieldbus : REFERENCE TO MachineFieldbus;
  _axis : REFERENCE TO MachineAxis;
  _data : REFERENCE TO MachineDataRef;
  _unit : REFERENCE TO MachineLinkedUnit;  
END_VAR

METHOD FB_init : BOOL
VAR_INPUT
  bInitRetains : BOOL; // if TRUE, the retain variables are initialized (warm start / cold start)
  bInCopyCode : BOOL;  // if TRUE, the instance afterwards gets moved into the copy code (online change)
  unit : REFERENCE TO MachineUnit;
END_VAR
_parent REF= unit;
_alarming := unit._alarming;
_io REF= unit._equipment.Io;
_actuator REF= unit._equipment.Actuator;
_fieldbus REF= unit._equipment.Fieldbus;
_axis REF= unit._equipment.Axis;
_unit REF= unit._equipment.Unit;
_data REF= unit._data;
_loggerDiagnostics.SetLogger(unit._logger);
END_METHOD

METHOD StepDecoded : ZCore.ZString
VAR_INPUT
  stepIndex : INT;
END_VAR
VAR_INST
  _stepIndexDecoded : MachineStep;
END_VAR
_stepIndexDecoded := stepIndex;
stepDecoded := TO_STRING(_stepIndexDecoded);
END_METHOD

END_FUNCTION_BLOCK

// ---- ZApp/Unit/Machine/_States/MachineSequenceAutomatic.TcPOU
FUNCTION_BLOCK MachineSequenceAutomatic EXTENDS MachineSequence IMPLEMENTS ZCore.ISequence
VAR
  _step : ZCore.Step(MachineStep.AutomaticBegin, MachineStep.AutomaticEnd);
  _timer : ZAux.Timer;
END_VAR

IF NOT Busy THEN
  RETURN;
END_IF

IF OnStart(_step) THEN
  ; // init custom sequence variables here ...
END_IF

IF OnStop() THEN
  RETURN; // external stop was triggered
END_IF

IF OnHalt() THEN
  Halting := TRUE;
END_IF

REPEAT
  LogStep();

  CASE _step.Index OF
    (* -------------------------------------------------------------------------------------------------------------------------------- *)
    MachineStep.AutomaticBegin:
    (* -------------------------------------------------------------------------------------------------------------------------------- *)
      IF _step.OnEntry()
      THEN
        _unit.PrimaryGear.RunAutomaticAsync(THIS^, _parent);
        _timer.WaitAsync(1);
      END_IF
      
      Assert(_unit.PrimaryGear);
      IF _unit.PrimaryGear.InSpeed AND_THEN _timer.Done
      THEN
        _step.SetNext(MachineStep.AutomaticAutomaticRunSecondaries);
			END_IF

    (* -------------------------------------------------------------------------------------------------------------------------------- *)
    MachineStep.AutomaticAutomaticRunSecondaries:
    (* -------------------------------------------------------------------------------------------------------------------------------- *)
      IF _step.OnEntry()
      THEN        
        _unit.SimpleGear.RunAutomaticAsync(THIS^, _parent);
        _unit.StruckigGear.RunAutomaticAsync(THIS^, _parent); 
      END_IF
         
      Await3(obj1:=_unit.PrimaryGear, obj2:=_unit.SimpleGear, obj3:=_unit.StruckigGear, nextStep:=MachineStep.AutomaticEnd);
      
    (* -------------------------------------------------------------------------------------------------------------------------------- *)
    MachineStep.AutomaticEnd:
    (* -------------------------------------------------------------------------------------------------------------------------------- *)
      SetBusy(FALSE);
  
  ELSE
    Abort('sequence contains unhandled step');
  END_CASE
UNTIL _step.IsNotRepeatable() OR_ELSE NOT Busy END_REPEAT

END_FUNCTION_BLOCK

// ---- ZApp/Unit/Machine/_States/MachineSequenceStop.TcPOU
FUNCTION_BLOCK MachineSequenceStop EXTENDS MachineSequence IMPLEMENTS ZCore.ISequence
VAR
  _step : ZCore.Step(MachineStep.StopBegin, MachineStep.StopEnd);
  _timerSim : ZAux.Timer;
END_VAR

IF OnStart(_step) THEN
  ; // init custom sequence variables here ...
END_IF

REPEAT
  LogStep();

  CASE _step.Index OF
    (* -------------------------------------------------------------------------------------------------------------------------------- *)
    MachineStep.StopBegin:
    (* -------------------------------------------------------------------------------------------------------------------------------- *)
      IF _step.OnEntry()
      THEN
        _unit.LeftGear.StopAsync(THIS^, _parent);
        _unit.RightGear.StopAsync(THIS^, _parent);        
      END_IF
      
      Await2(_unit.LeftGear, _unit.RightGear, nextStep:=MachineStep.StopEnd);

    (* -------------------------------------------------------------------------------------------------------------------------------- *)
    MachineStep.StopEnd:
    (* -------------------------------------------------------------------------------------------------------------------------------- *)    
      SetBusy(FALSE);
  
  ELSE
    Abort('sequence contains unhandled step');
  END_CASE
UNTIL _step.IsNotRepeatable() OR_ELSE NOT Busy END_REPEAT

END_FUNCTION_BLOCK

// ---- ZApp/Unit/Machine/_States/MachineSequenceGoHome.TcPOU
FUNCTION_BLOCK MachineSequenceGoHome EXTENDS MachineSequence IMPLEMENTS ZCore.ISequence
VAR
  _step : ZCore.Step(MachineStep.GohomeBegin, MachineStep.GohomeEnd);
  _timer : ZAux.Timer;
END_VAR

IF NOT Busy THEN
  RETURN;
END_IF

IF OnStart(_step) THEN
  ; // init custom sequence variables here ...
END_IF

IF OnStop() THEN
  RETURN; // external stop was triggered
END_IF

IF OnHalt() THEN
  ; // Halting := TRUE; // Uncomment to acknowledge that the sequence is halting
END_IF

REPEAT
  LogStep();

  CASE _step.Index OF
    (* -------------------------------------------------------------------------------------------------------------------------------- *)
    MachineStep.GoHomeBegin:
    (* -------------------------------------------------------------------------------------------------------------------------------- *)
      IF _step.OnEntry()
      THEN
        _unit.PrimaryGear.HomingAsync(THIS^, _parent);
        _timer.WaitAsync(3);
      END_IF
      
      Await2(_unit.PrimaryGear, _timer, nextStep:=MachineStep.GoHomeGoHomeSecondaries);

    (* -------------------------------------------------------------------------------------------------------------------------------- *)
    MachineStep.GoHomeGoHomeSecondaries:
    (* -------------------------------------------------------------------------------------------------------------------------------- *)
      IF _step.OnEntry()
      THEN        
        _unit.SimpleGear.HomingAsync(THIS^, _parent);
        _unit.StruckigGear.HomingAsync(THIS^, _parent);   
      END_IF
      
      Await2(_unit.SimpleGear, _unit.StruckigGear, nextStep:=MachineStep.GoHomeEnd);

    (* -------------------------------------------------------------------------------------------------------------------------------- *)
    MachineStep.GoHomeEnd:
    (* -------------------------------------------------------------------------------------------------------------------------------- *)
      SetBusy(FALSE);
  
  ELSE
    Abort('sequence contains unhandled step');
  END_CASE
UNTIL _step.IsNotRepeatable() OR_ELSE NOT Busy END_REPEAT

END_FUNCTION_BLOCK

// ---- ZApp/Unit/Machine/_States/MachineSequenceFaultReaction.TcPOU
FUNCTION_BLOCK MachineSequenceFaultReaction EXTENDS MachineSequence IMPLEMENTS ZCore.ISequence
VAR
  _step : ZCore.Step(MachineStep.FaultReactionBegin, MachineStep.FaultReactionEnd);
  _timerSim : ZAux.Timer;
END_VAR

IF OnStart(_step) THEN
  ; // init custom sequence variables here ...
END_IF

REPEAT
  LogStep();

  CASE _step.Index OF
    (* -------------------------------------------------------------------------------------------------------------------------------- *)
    MachineStep.FaultReactionBegin:
    (* -------------------------------------------------------------------------------------------------------------------------------- *)
      IF _step.OnEntry()
      THEN
        _unit.PrimaryGear.StopAsync(THIS^, _parent);
        _unit.SimpleGear.StopAsync(THIS^, _parent);    
        _unit.StruckigGear.StopAsync(THIS^, _parent);        
      END_IF
      
      _step.SetNext(MachineStep.FaultReactionEnd);

    (* -------------------------------------------------------------------------------------------------------------------------------- *)
    MachineStep.FaultReactionEnd:
    (* -------------------------------------------------------------------------------------------------------------------------------- *)    
      SetBusy(FALSE);
  
  ELSE
    Abort('sequence contains unhandled step');
  END_CASE
UNTIL _step.IsNotRepeatable() OR_ELSE NOT Busy END_REPEAT

END_FUNCTION_BLOCK

// ---- ZApp/Unit/Gear/GearUnitProgram.TcPOU
/// each unit can run in its own PROGRAM and Task, respectively. However, this is optional and one may also
/// instantiate the unit in the ModuleProgram.
/// In order to keep initialization to a minimum, all ModuleContext objects that are required by the Unit are
/// given as FB_init parameter. These objects are
/// * data structs
/// * communication structs
/// * busmaster(s)
/// A unit should always be a root object (no parent) if it is running in its own context. If it runs in the same
/// task as the Module the parent may be set to the Module's Application.
PROGRAM GearUnitProgram
VAR
{region "PrimaryGear"}
{undefine RunInSeparateProgram}
{IF NOT (defined (PrimaryGear_disabled)) AND (defined (RunInSeparateProgram))}
  PrimaryGear : GearUnit(name := 'PrimaryGear', // name of the unit (for logging)
					  parent := 0, // caller of the Unit's cyclic method. If the Unit runs in its own context use 0
						configdata := ZGlobal.Data.Config.PrimaryGear,
						machinedata := ZGlobal.Data.Machine.PrimaryGear,
						calibrationdata := ZGlobal.Data.Calibration.PrimaryGear,
						com := ZGlobal.Com.Unit.PrimaryGear);
  {attribute 'section' := '__ZwPlcUnitProgramDeclaration__'}
  {attribute 'ZId' := 'd1deea68-6f8b-4ea5-9916-7be69dc951fa'}
{END_IF}
{endregion}
{region "SimpleGear"}
{undefine RunInSeparateProgram}
{IF NOT (defined (SimpleGear_disabled)) AND (defined (RunInSeparateProgram))}
  SimpleGear : GearUnit(name := 'SimpleGear', // name of the unit (for logging)
					  parent := 0, // caller of the Unit's cyclic method. If the Unit runs in its own context use 0
						configdata := ZGlobal.Data.Config.SimpleGear,
						machinedata := ZGlobal.Data.Machine.SimpleGear,
						calibrationdata := ZGlobal.Data.Calibration.SimpleGear,
						com := ZGlobal.Com.Unit.SimpleGear);
  {attribute 'section' := '__ZwPlcUnitProgramDeclaration__'}
  {attribute 'ZId' := '215d1db4-d61a-4f46-91b5-612373b86c91'}
{END_IF}
{endregion}
{region "StruckigGear"}
{undefine RunInSeparateProgram}
{IF NOT (defined (StruckigGear_disabled)) AND (defined (RunInSeparateProgram))}
  StruckigGear : GearUnit(name := 'StruckigGear', // name of the unit (for logging)
					  parent := 0, // caller of the Unit's cyclic method. If the Unit runs in its own context use 0
						configdata := ZGlobal.Data.Config.StruckigGear,
						machinedata := ZGlobal.Data.Machine.StruckigGear,
						calibrationdata := ZGlobal.Data.Calibration.StruckigGear,
						com := ZGlobal.Com.Unit.StruckigGear);
  {attribute 'section' := '__ZwPlcUnitProgramDeclaration__'}
  {attribute 'ZId' := 'd827270e-999f-436d-80d5-b12442f5d1cf'}
{END_IF}
{endregion}
{attribute '__ZwPlcUnitProgramDeclaration__'} // Do not remove this attribute! It is used for code generation.
END_VAR

// run the unit - the cylics of all children will be called as well

{region "PrimaryGear"}
{undefine RunInSeparateProgram}
{IF NOT (defined (PrimaryGear_disabled)) AND (defined (RunInSeparateProgram))}
  PrimaryGear.Cyclic();
  {attribute 'section' := '__ZwPlcUnitProgramImplementation__'}
  {attribute 'ZId' := 'd1deea68-6f8b-4ea5-9916-7be69dc951fa'}
{END_IF}
{endregion}
{region "SimpleGear"}
{undefine RunInSeparateProgram}
{IF NOT (defined (SimpleGear_disabled)) AND (defined (RunInSeparateProgram))}
  SimpleGear.Cyclic();
  {attribute 'section' := '__ZwPlcUnitProgramImplementation__'}
  {attribute 'ZId' := '215d1db4-d61a-4f46-91b5-612373b86c91'}
{END_IF}
{endregion}
{region "StruckigGear"}
{undefine RunInSeparateProgram}
{IF NOT (defined (StruckigGear_disabled)) AND (defined (RunInSeparateProgram))}
  StruckigGear.Cyclic();
  {attribute 'section' := '__ZwPlcUnitProgramImplementation__'}
  {attribute 'ZId' := 'd827270e-999f-436d-80d5-b12442f5d1cf'}
{END_IF}
{endregion}
{attribute '__ZwPlcUnitProgramImplementation__'} // Do not remove this attribute! It is used for code generation.

END_PROGRAM

// ---- ZApp/Unit/Machine/MachineUnitProgram.TcPOU
/// each unit can run in its own PROGRAM and Task, respectively. However, this is optional and one may also
/// instantiate the unit in the ModuleProgram.
/// In order to keep initialization to a minimum, all ModuleContext objects that are required by the Unit are
/// given as FB_init parameter. These objects are
/// * data structs
/// * communication structs
/// * busmaster(s)
/// A unit should always be a root object (no parent) if it is running in its own context. If it runs in the same
/// task as the Module the parent may be set to the Module's Application.
PROGRAM MachineUnitProgram
VAR
{region "Machine"}
{undefine RunInSeparateProgram}
{IF NOT (defined (Machine_disabled)) AND (defined (RunInSeparateProgram))}
  Machine : MachineUnit(name := 'Machine', // name of the unit (for logging)
					  parent := 0, // caller of the Unit's cyclic method. If the Unit runs in its own context use 0
						configdata := ZGlobal.Data.Config.Machine,
						machinedata := ZGlobal.Data.Machine.Machine,
						calibrationdata := ZGlobal.Data.Calibration.Machine,
						com := ZGlobal.Com.Unit.Machine);
  {attribute 'section' := '__ZwPlcUnitProgramDeclaration__'}
  {attribute 'ZId' := '9a1e8940-043c-4b8f-bd95-526fb267b71c'}
{END_IF}
{endregion}
{attribute '__ZwPlcUnitProgramDeclaration__'} // Do not remove this attribute! It is used for code generation.
END_VAR

// run the unit - the cylics of all children will be called as well

{region "Machine"}
{undefine RunInSeparateProgram}
{IF NOT (defined (Machine_disabled)) AND (defined (RunInSeparateProgram))}
  Machine.Cyclic();
  {attribute 'section' := '__ZwPlcUnitProgramImplementation__'}
  {attribute 'ZId' := '9a1e8940-043c-4b8f-bd95-526fb267b71c'}
{END_IF}
{endregion}
{attribute '__ZwPlcUnitProgramImplementation__'} // Do not remove this attribute! It is used for code generation.

END_PROGRAM
